LIN {X 0,Y 220.797,Z 443.981,A -85,B 0,C 180,E1 -20381.946,E2 -20381.946} C_VEL
LIN {X 0,Y 220.875,Z 443.967,A -85,B 0,C 180,E1 -20387.041,E2 -20387.041} C_VEL
LIN {X 0,Y 220.861,Z 443.966,A -85,B 0,C 180,E1 -20390.474,E2 -20390.474} C_VEL
LIN {X 0,Y 220.818,Z 443.975,A -85,B 0,C 180,E1 -20395.048,E2 -20395.048} C_VEL
LIN {X 0,Y 220.906,Z 444.135,A -85,B 0,C 180,E1 -20396.999,E2 -20396.999} C_VEL
LIN {X 0,Y 221.881,Z 446.769,A -85,B 0,C 180,E1 -20397.42,E2 -20397.42} C_VEL
LIN {X 0,Y 226.651,Z 456.679,A -85,B 0,C 180,E1 -20399.386,E2 -20399.386} C_VEL
LIN {X 0,Y 230.145,Z 465.491,A -85,B 0,C 180,E1 -20401.214,E2 -20401.214} C_VEL
LIN {X 0,Y 233.063,Z 475.055,A -85,B 0,C 180,E1 -20403.323,E2 -20403.323} C_VEL
LIN {X 0,Y 234.867,Z 483.039,A -85,B 0,C 180,E1 -20405.233,E2 -20405.233} C_VEL
LIN {X 0,Y 232.591,Z 492.857,A -85,B 0,C 180,E1 -20407.34,E2 -20407.34} C_VEL
LIN {X 0,Y 230.039,Z 502.346,A -85,B 0,C 180,E1 -20409.897,E2 -20409.897} C_VEL
LIN {X 0,Y 227.751,Z 509.911,A -85,B 0,C 180,E1 -20412.49,E2 -20412.49} C_VEL
LIN {X 0,Y 226.25,Z 515.061,A -85,B 0,C 180,E1 -20414.7,E2 -20414.7} C_VEL
LIN {X 0,Y 224.746,Z 520.013,A -85,B 0,C 180,E1 -20417.356,E2 -20417.356} C_VEL
LIN {X 0,Y 223.377,Z 523.89,A -85,B 0,C 180,E1 -20420.035,E2 -20420.035} C_VEL
LIN {X 0,Y 222.303,Z 526.757,A -85,B 0,C 180,E1 -20422.735,E2 -20422.735} C_VEL
LIN {X 0,Y 221.792,Z 528.126,A -85,B 0,C 180,E1 -20424.545,E2 -20424.545} C_VEL
LIN {X 0,Y 221.55,Z 529.649,A -85,B 0,C 180,E1 -20428.182,E2 -20428.182} C_VEL
LIN {X 0,Y 221.511,Z 529.869,A -85,B 0,C 180,E1 -20430,E2 -20430} C_VEL
LIN {X 0,Y 221.549,Z 529.683,A -85,B 0,C 180,E1 -20431.818,E2 -20431.818} C_VEL
LIN {X 0,Y 221.782,Z 528.204,A -85,B 0,C 180,E1 -20435.455,E2 -20435.455} C_VEL
LIN {X 0,Y 222.287,Z 526.871,A -85,B 0,C 180,E1 -20437.265,E2 -20437.265} C_VEL
LIN {X 0,Y 223.365,Z 524.046,A -85,B 0,C 180,E1 -20439.965,E2 -20439.965} C_VEL
LIN {X 0,Y 224.708,Z 520.225,A -85,B 0,C 180,E1 -20442.646,E2 -20442.646} C_VEL
LIN {X 0,Y 226.414,Z 514.308,A -85,B 0,C 180,E1 -20445.791,E2 -20445.791} C_VEL
LIN {X 0,Y 228.461,Z 507.907,A -85,B 0,C 180,E1 -20448.38,E2 -20448.38} C_VEL
LIN {X 0,Y 230.832,Z 499.865,A -85,B 0,C 180,E1 -20450.962,E2 -20450.962} C_VEL
LIN {X 0,Y 232.897,Z 491.636,A -85,B 0,C 180,E1 -20453.097,E2 -20453.097} C_VEL
LIN {X 0,Y 234.818,Z 483.666,A -85,B 0,C 180,E1 -20454.772,E2 -20454.772} C_VEL
LIN {X 0,Y 234.22,Z 479.238,A -85,B 0,C 180,E1 -20455.818,E2 -20455.818} C_VEL
LIN {X 0,Y 231.252,Z 468.913,A -85,B 0,C 180,E1 -20458.195,E2 -20458.195} C_VEL
LIN {X 0,Y 227.759,Z 459.239,A -85,B 0,C 180,E1 -20460.231,E2 -20460.231} C_VEL
LIN {X 0,Y 222.646,Z 448.097,A -85,B 0,C 180,E1 -20462.454,E2 -20462.454} C_VEL
LIN {X 0,Y 220.923,Z 444.348,A -85,B 0,C 180,E1 -20463.132,E2 -20463.132} C_VEL
LIN {X 0,Y 220.874,Z 443.97,A -85,B 0,C 180,E1 -20463.221,E2 -20463.221} C_VEL
LIN {X 0,Y 220.869,Z 443.973,A -85,B 0,C 180,E1 -20467.298,E2 -20467.298} C_VEL
LIN {X 0,Y 220.873,Z 443.971,A -85,B 0,C 180,E1 -20471.929,E2 -20471.929} C_VEL
LIN {X 0,Y 220.792,Z 443.981,A -85,B 0,C 180,E1 -20475.55,E2 -20475.55} C_VEL
LIN {X 0,Y 220.811,Z 443.98,A -85,B 0,C 180,E1 -20480.464,E2 -20480.464} C_VEL
LIN {X 0,Y 220.802,Z 443.984,A -85,B 0,C 180,E1 -20485.045,E2 -20485.045} C_VEL
LIN {X 0,Y 220.835,Z 443.977,A -85,B 0,C 180,E1 -20489.39,E2 -20489.39} C_VEL
LIN {X 0,Y 220.896,Z 443.967,A -85,B 0,C 180,E1 -20493.549,E2 -20493.549} C_VEL
LIN {X 0,Y 220.88,Z 443.963,A -85,B 0,C 180,E1 -20497.553,E2 -20497.553} C_VEL
LIN {X 0,Y 220.986,Z 443.952,A -85,B 0,C 180,E1 -20502.571,E2 -20502.571} C_VEL
LIN {X 0,Y 221.014,Z 443.95,A -85,B 0,C 180,E1 -20507.139,E2 -20507.139} C_VEL
LIN {X 0,Y 221.204,Z 443.931,A -85,B 0,C 180,E1 -20510.859,E2 -20510.859} C_VEL
LIN {X 0,Y 221.14,Z 443.925,A -85,B 0,C 180,E1 -20514.529,E2 -20514.529} C_VEL
LIN {X 0,Y 221.515,Z 443.892,A -85,B 0,C 180,E1 -20518.182,E2 -20518.182} C_VEL
LIN {X 0,Y 221.515,Z 443.88,A -85,B 0,C 180,E1 -20521.818,E2 -20521.818} C_VEL
LIN {X 0,Y 221.257,Z 443.916,A -85,B 0,C 180,E1 -20527.299,E2 -20527.299} C_VEL
LIN {X 0,Y 221.083,Z 443.944,A -85,B 0,C 180,E1 -20530.996,E2 -20530.996} C_VEL
LIN {X 0,Y 221.018,Z 443.949,A -85,B 0,C 180,E1 -20536.63,E2 -20536.63} C_VEL
LIN {X 0,Y 220.886,Z 443.973,A -85,B 0,C 180,E1 -20540.487,E2 -20540.487} C_VEL
LIN {X 0,Y 220.863,Z 443.975,A -85,B 0,C 180,E1 -20544.435,E2 -20544.435} C_VEL
LIN {X 0,Y 220.828,Z 443.978,A -85,B 0,C 180,E1 -20548.515,E2 -20548.515} C_VEL
LIN {X 0,Y 220.83,Z 444.003,A -85,B 0,C 180,E1 -20551.675,E2 -20551.675} C_VEL
LIN {X 0,Y 221.956,Z 449.045,A -85,B 0,C 180,E1 -20555.858,E2 -20555.858} C_VEL
LIN {X 0,Y 223.004,Z 454.546,A -85,B 0,C 180,E1 -20560.02,E2 -20560.02} C_VEL
LIN {X 0,Y 224.02,Z 459.907,A -85,B 0,C 180,E1 -20563.816,E2 -20563.816} C_VEL
LIN {X 0,Y 225.122,Z 465.25,A -85,B 0,C 180,E1 -20567.382,E2 -20567.382} C_VEL
LIN {X 0,Y 225.601,Z 467.977,A -85,B 0,C 180,E1 -20569.141,E2 -20569.141} C_VEL
LIN {X 0,Y 225.692,Z 469.86,A -85,B 0,C 180,E1 -20570.314,E2 -20570.314} C_VEL
LIN {X 0,Y 224.095,Z 476.513,A -85,B 0,C 180,E1 -20574.172,E2 -20574.172} C_VEL
LIN {X 0,Y 223.25,Z 479.952,A -85,B 0,C 180,E1 -20576.149,E2 -20576.149} C_VEL
LIN {X 0,Y 224.695,Z 487.159,A -85,B 0,C 180,E1 -20576.76,E2 -20576.76} C_VEL
LIN {X 0,Y 226.787,Z 499.616,A -85,B 0,C 180,E1 -20577.987,E2 -20577.987} C_VEL
LIN {X 0,Y 228.055,Z 512.378,A -85,B 0,C 180,E1 -20579.46,E2 -20579.46} C_VEL
LIN {X 0,Y 228.416,Z 525.424,A -85,B 0,C 180,E1 -20581.265,E2 -20581.265} C_VEL
LIN {X 0,Y 228.421,Z 526.853,A -85,B 0,C 180,E1 -20581.483,E2 -20581.483} C_VEL
LIN {X 0,Y 227.726,Z 531.904,A -85,B 0,C 180,E1 -20582.228,E2 -20582.228} C_VEL
LIN {X 0,Y 225.999,Z 536.833,A -85,B 0,C 180,E1 -20582.945,E2 -20582.945} C_VEL
LIN {X 0,Y 220.98,Z 547.697,A -85,B 0,C 180,E1 -20584.798,E2 -20584.798} C_VEL
LIN {X 0,Y 219.703,Z 552.067,A -85,B 0,C 180,E1 -20585.794,E2 -20585.794} C_VEL
LIN {X 0,Y 218.356,Z 559.465,A -85,B 0,C 180,E1 -20587.779,E2 -20587.779} C_VEL
LIN {X 0,Y 215.907,Z 568.5,A -85,B 0,C 180,E1 -20590.732,E2 -20590.732} C_VEL
LIN {X 0,Y 214.238,Z 574.791,A -85,B 0,C 180,E1 -20593.319,E2 -20593.319} C_VEL
LIN {X 0,Y 213.015,Z 581.157,A -85,B 0,C 180,E1 -20596.647,E2 -20596.647} C_VEL
LIN {X 0,Y 212.567,Z 585.353,A -85,B 0,C 180,E1 -20599.523,E2 -20599.523} C_VEL
LIN {X 0,Y 212.669,Z 588.586,A -85,B 0,C 180,E1 -20602.481,E2 -20602.481} C_VEL
LIN {X 0,Y 213.218,Z 591.167,A -85,B 0,C 180,E1 -20606.22,E2 -20606.22} C_VEL
LIN {X 0,Y 213.999,Z 592.157,A -85,B 0,C 180,E1 -20610,E2 -20610} C_VEL
LIN {X 0,Y 213.215,Z 591.15,A -85,B 0,C 180,E1 -20613.78,E2 -20613.78} C_VEL
LIN {X 0,Y 212.627,Z 588.624,A -85,B 0,C 180,E1 -20617.432,E2 -20617.432} C_VEL
LIN {X 0,Y 212.568,Z 585.304,A -85,B 0,C 180,E1 -20620.477,E2 -20620.477} C_VEL
LIN {X 0,Y 213.014,Z 581.088,A -85,B 0,C 180,E1 -20623.353,E2 -20623.353} C_VEL
LIN {X 0,Y 214.21,Z 574.691,A -85,B 0,C 180,E1 -20626.683,E2 -20626.683} C_VEL
LIN {X 0,Y 215.907,Z 568.382,A -85,B 0,C 180,E1 -20629.269,E2 -20629.269} C_VEL
LIN {X 0,Y 218.348,Z 559.319,A -85,B 0,C 180,E1 -20632.222,E2 -20632.222} C_VEL
LIN {X 0,Y 219.865,Z 550.517,A -85,B 0,C 180,E1 -20634.554,E2 -20634.554} C_VEL
LIN {X 0,Y 221.04,Z 540.018,A -85,B 0,C 180,E1 -20636.856,E2 -20636.856} C_VEL
LIN {X 0,Y 221.682,Z 528.784,A -85,B 0,C 180,E1 -20638.913,E2 -20638.913} C_VEL
LIN {X 0,Y 221.703,Z 517.176,A -85,B 0,C 180,E1 -20640.699,E2 -20640.699} C_VEL
LIN {X 0,Y 220.89,Z 504.818,A -85,B 0,C 180,E1 -20642.312,E2 -20642.312} C_VEL
LIN {X 0,Y 219.065,Z 491.67,A -85,B 0,C 180,E1 -20643.777,E2 -20643.777} C_VEL
LIN {X 0,Y 216.635,Z 478.749,A -85,B 0,C 180,E1 -20645.03,E2 -20645.03} C_VEL
LIN {X 0,Y 218.558,Z 471.281,A -85,B 0,C 180,E1 -20649.489,E2 -20649.489} C_VEL
LIN {X 0,Y 218.545,Z 468.802,A -85,B 0,C 180,E1 -20651.076,E2 -20651.076} C_VEL
LIN {X 0,Y 217.309,Z 462.5,A -85,B 0,C 180,E1 -20655.358,E2 -20655.358} C_VEL
LIN {X 0,Y 216.224,Z 456.823,A -85,B 0,C 180,E1 -20659.453,E2 -20659.453} C_VEL
LIN {X 0,Y 215.145,Z 450.979,A -85,B 0,C 180,E1 -20663.985,E2 -20663.985} C_VEL
LIN {X 0,Y 213.875,Z 445.272,A -85,B 0,C 180,E1 -20668.917,E2 -20668.917} C_VEL
LIN {X 0,Y 213.779,Z 444.857,A -85,B 0,C 180,E1 -20669.56,E2 -20669.56} C_VEL
LIN {X 0,Y 213.828,Z 444.855,A -85,B 0,C 180,E1 -20672.604,E2 -20672.604} C_VEL
LIN {X 0,Y 213.822,Z 444.849,A -85,B 0,C 180,E1 -20676.974,E2 -20676.974} C_VEL
LIN {X 0,Y 213.947,Z 444.836,A -85,B 0,C 180,E1 -20682.804,E2 -20682.804} C_VEL
LIN {X 0,Y 213.957,Z 444.837,A -85,B 0,C 180,E1 -20686.707,E2 -20686.707} C_VEL
LIN {X 0,Y 214.142,Z 444.811,A -85,B 0,C 180,E1 -20690.555,E2 -20690.555} C_VEL
LIN {X 0,Y 214.103,Z 444.817,A -85,B 0,C 180,E1 -20694.349,E2 -20694.349} C_VEL
LIN {X 0,Y 214.45,Z 444.774,A -85,B 0,C 180,E1 -20698.122,E2 -20698.122} C_VEL
LIN {X 0,Y 214.558,Z 444.757,A -85,B 0,C 180,E1 -20700,E2 -20700} C_VEL
LIN {X 0,Y 214.449,Z 444.773,A -85,B 0,C 180,E1 -20701.878,E2 -20701.878} C_VEL
LIN {X 0,Y 214.197,Z 444.802,A -85,B 0,C 180,E1 -20707.542,E2 -20707.542} C_VEL
LIN {X 0,Y 214.011,Z 444.816,A -85,B 0,C 180,E1 -20711.364,E2 -20711.364} C_VEL
LIN {X 0,Y 213.936,Z 444.787,A -85,B 0,C 180,E1 -20715.237,E2 -20715.237} C_VEL
LIN {X 0,Y 213.843,Z 444.831,A -85,B 0,C 180,E1 -20719.187,E2 -20719.187} C_VEL
LIN {X 0,Y 213.85,Z 444.841,A -85,B 0,C 180,E1 -20723.227,E2 -20723.227} C_VEL
LIN {X 0,Y 213.832,Z 444.809,A -85,B 0,C 180,E1 -20727.45,E2 -20727.45} C_VEL
LIN {X 0,Y 213.77,Z 444.852,A -85,B 0,C 180,E1 -20731.737,E2 -20731.737} C_VEL
LIN {X 0,Y 213.746,Z 444.855,A -85,B 0,C 180,E1 -20736.288,E2 -20736.288} C_VEL
LIN {X 0,Y 213.728,Z 444.861,A -85,B 0,C 180,E1 -20741.122,E2 -20741.122} C_VEL
LIN {X 0,Y 213.75,Z 444.854,A -85,B 0,C 180,E1 -20743.668,E2 -20743.668} C_VEL
LIN {X 0,Y 213.814,Z 444.85,A -85,B 0,C 180,E1 -20746.349,E2 -20746.349} C_VEL
LIN {X 0,Y 213.8,Z 444.851,A -85,B 0,C 180,E1 -20749.118,E2 -20749.118} C_VEL
LIN {X 0,Y 213.759,Z 444.849,A -85,B 0,C 180,E1 -20753.714,E2 -20753.714} C_VEL
LIN {X 0,Y 213.799,Z 445.01,A -85,B 0,C 180,E1 -20755.719,E2 -20755.719} C_VEL
LIN {X 0,Y 214.42,Z 446.987,A -85,B 0,C 180,E1 -20756.032,E2 -20756.032} C_VEL
LIN {X 0,Y 215.693,Z 448.943,A -85,B 0,C 180,E1 -20756.485,E2 -20756.485} C_VEL
LIN {X 0,Y 220.507,Z 459.407,A -85,B 0,C 180,E1 -20758.674,E2 -20758.674} C_VEL
LIN {X 0,Y 224.284,Z 469.275,A -85,B 0,C 180,E1 -20760.865,E2 -20760.865} C_VEL
LIN {X 0,Y 227.226,Z 479.67,A -85,B 0,C 180,E1 -20763.327,E2 -20763.327} C_VEL
LIN {X 0,Y 228.28,Z 485.103,A -85,B 0,C 180,E1 -20764.712,E2 -20764.712} C_VEL
LIN {X 0,Y 226.124,Z 493.865,A -85,B 0,C 180,E1 -20766.654,E2 -20766.654} C_VEL
LIN {X 0,Y 223.452,Z 503.353,A -85,B 0,C 180,E1 -20769.278,E2 -20769.278} C_VEL
LIN {X 0,Y 221.059,Z 510.918,A -85,B 0,C 180,E1 -20771.942,E2 -20771.942} C_VEL
LIN {X 0,Y 219.481,Z 516.063,A -85,B 0,C 180,E1 -20774.213,E2 -20774.213} C_VEL
LIN {X 0,Y 217.895,Z 521.019,A -85,B 0,C 180,E1 -20776.951,E2 -20776.951} C_VEL
LIN {X 0,Y 216.458,Z 524.896,A -85,B 0,C 180,E1 -20779.713,E2 -20779.713} C_VEL
LIN {X 0,Y 215.333,Z 527.763,A -85,B 0,C 180,E1 -20782.498,E2 -20782.498} C_VEL
LIN {X 0,Y 214.797,Z 529.132,A -85,B 0,C 180,E1 -20784.367,E2 -20784.367} C_VEL
LIN {X 0,Y 214.526,Z 530.654,A -85,B 0,C 180,E1 -20788.122,E2 -20788.122} C_VEL
LIN {X 0,Y 214.484,Z 530.874,A -85,B 0,C 180,E1 -20790,E2 -20790} C_VEL
LIN {X 0,Y 214.525,Z 530.687,A -85,B 0,C 180,E1 -20791.877,E2 -20791.877} C_VEL
LIN {X 0,Y 214.787,Z 529.209,A -85,B 0,C 180,E1 -20795.633,E2 -20795.633} C_VEL
LIN {X 0,Y 215.317,Z 527.875,A -85,B 0,C 180,E1 -20797.502,E2 -20797.502} C_VEL
LIN {X 0,Y 216.446,Z 525.05,A -85,B 0,C 180,E1 -20800.287,E2 -20800.287} C_VEL
LIN {X 0,Y 217.856,Z 521.229,A -85,B 0,C 180,E1 -20803.051,E2 -20803.051} C_VEL
LIN {X 0,Y 219.658,Z 515.315,A -85,B 0,C 180,E1 -20806.288,E2 -20806.288} C_VEL
LIN {X 0,Y 221.803,Z 508.91,A -85,B 0,C 180,E1 -20808.952,E2 -20808.952} C_VEL
LIN {X 0,Y 224.283,Z 500.868,A -85,B 0,C 180,E1 -20811.604,E2 -20811.604} C_VEL
LIN {X 0,Y 226.451,Z 492.638,A -85,B 0,C 180,E1 -20813.795,E2 -20813.795} C_VEL
LIN {X 0,Y 228.303,Z 484.691,A -85,B 0,C 180,E1 -20815.529,E2 -20815.529} C_VEL
LIN {X 0,Y 226.822,Z 477.955,A -85,B 0,C 180,E1 -20817.232,E2 -20817.232} C_VEL
LIN {X 0,Y 224.28,Z 469.314,A -85,B 0,C 180,E1 -20819.278,E2 -20819.278} C_VEL
LIN {X 0,Y 220.91,Z 460.371,A -85,B 0,C 180,E1 -20821.272,E2 -20821.272} C_VEL
LIN {X 0,Y 215.802,Z 449.254,A -85,B 0,C 180,E1 -20823.617,E2 -20823.617} C_VEL
LIN {X 0,Y 213.944,Z 445.703,A -85,B 0,C 180,E1 -20824.345,E2 -20824.345} C_VEL
LIN {X 0,Y 213.773,Z 444.851,A -85,B 0,C 180,E1 -20824.476,E2 -20824.476} C_VEL
LIN {X 0,Y 213.805,Z 444.853,A -85,B 0,C 180,E1 -20828.649,E2 -20828.649} C_VEL
LIN {X 0,Y 213.829,Z 444.851,A -85,B 0,C 180,E1 -20831.098,E2 -20831.098} C_VEL
LIN {X 0,Y 213.81,Z 444.851,A -85,B 0,C 180,E1 -20833.685,E2 -20833.685} C_VEL
LIN {X 0,Y 213.749,Z 444.86,A -85,B 0,C 180,E1 -20836.332,E2 -20836.332} C_VEL
LIN {X 0,Y 213.727,Z 444.863,A -85,B 0,C 180,E1 -20841.334,E2 -20841.334} C_VEL
LIN {X 0,Y 213.758,Z 444.859,A -85,B 0,C 180,E1 -20846.018,E2 -20846.018} C_VEL
LIN {X 0,Y 213.762,Z 444.86,A -85,B 0,C 180,E1 -20850.451,E2 -20850.451} C_VEL
LIN {X 0,Y 213.803,Z 444.854,A -85,B 0,C 180,E1 -20854.702,E2 -20854.702} C_VEL
LIN {X 0,Y 213.815,Z 444.848,A -85,B 0,C 180,E1 -20858.803,E2 -20858.803} C_VEL
LIN {X 0,Y 213.946,Z 444.828,A -85,B 0,C 180,E1 -20862.804,E2 -20862.804} C_VEL
LIN {X 0,Y 213.956,Z 444.831,A -85,B 0,C 180,E1 -20866.707,E2 -20866.707} C_VEL
LIN {X 0,Y 214.142,Z 444.811,A -85,B 0,C 180,E1 -20870.555,E2 -20870.555} C_VEL
LIN {X 0,Y 214.1,Z 444.802,A -85,B 0,C 180,E1 -20874.348,E2 -20874.348} C_VEL
LIN {X 0,Y 214.448,Z 444.772,A -85,B 0,C 180,E1 -20878.122,E2 -20878.122} C_VEL
LIN {X 0,Y 214.557,Z 444.756,A -85,B 0,C 180,E1 -20880,E2 -20880} C_VEL
LIN {X 0,Y 214.448,Z 444.76,A -85,B 0,C 180,E1 -20881.878,E2 -20881.878} C_VEL
LIN {X 0,Y 214.196,Z 444.794,A -85,B 0,C 180,E1 -20887.541,E2 -20887.541} C_VEL
LIN {X 0,Y 214.01,Z 444.825,A -85,B 0,C 180,E1 -20891.364,E2 -20891.364} C_VEL
LIN {X 0,Y 213.936,Z 444.836,A -85,B 0,C 180,E1 -20895.237,E2 -20895.237} C_VEL
LIN {X 0,Y 213.838,Z 444.849,A -85,B 0,C 180,E1 -20899.187,E2 -20899.187} C_VEL
LIN {X 0,Y 213.812,Z 444.852,A -85,B 0,C 180,E1 -20903.231,E2 -20903.231} C_VEL
LIN {X 0,Y 213.83,Z 444.85,A -85,B 0,C 180,E1 -20907.45,E2 -20907.45} C_VEL
LIN {X 0,Y 213.81,Z 445.01,A -85,B 0,C 180,E1 -20910.769,E2 -20910.769} C_VEL
LIN {X 0,Y 214.585,Z 448.483,A -85,B 0,C 180,E1 -20913.833,E2 -20913.833} C_VEL
LIN {X 0,Y 215.7,Z 453.941,A -85,B 0,C 180,E1 -20918.248,E2 -20918.248} C_VEL
LIN {X 0,Y 216.85,Z 460.139,A -85,B 0,C 180,E1 -20922.891,E2 -20922.891} C_VEL
LIN {X 0,Y 218.259,Z 467.186,A -85,B 0,C 180,E1 -20927.783,E2 -20927.783} C_VEL
LIN {X 0,Y 218.664,Z 470.579,A -85,B 0,C 180,E1 -20929.998,E2 -20929.998} C_VEL
LIN {X 0,Y 217.389,Z 475.884,A -85,B 0,C 180,E1 -20933.204,E2 -20933.204} C_VEL
LIN {X 0,Y 216.645,Z 478.821,A -85,B 0,C 180,E1 -20934.965,E2 -20934.965} C_VEL
LIN {X 0,Y 219.458,Z 493.611,A -85,B 0,C 180,E1 -20936.37,E2 -20936.37} C_VEL
LIN {X 0,Y 221.046,Z 505.767,A -85,B 0,C 180,E1 -20937.754,E2 -20937.754} C_VEL
LIN {X 0,Y 221.758,Z 517.676,A -85,B 0,C 180,E1 -20939.327,E2 -20939.327} C_VEL
LIN {X 0,Y 221.762,Z 529.086,A -85,B 0,C 180,E1 -20941.099,E2 -20941.099} C_VEL
LIN {X 0,Y 221.056,Z 540.207,A -85,B 0,C 180,E1 -20943.136,E2 -20943.136} C_VEL
LIN {X 0,Y 219.923,Z 550.713,A -85,B 0,C 180,E1 -20945.453,E2 -20945.453} C_VEL
LIN {X 0,Y 219.703,Z 552.067,A -85,B 0,C 180,E1 -20945.794,E2 -20945.794} C_VEL
LIN {X 0,Y 218.282,Z 556.263,A -85,B 0,C 180,E1 -20946.832,E2 -20946.832} C_VEL
LIN {X 0,Y 215.837,Z 560.132,A -85,B 0,C 180,E1 -20947.837,E2 -20947.837} C_VEL
LIN {X 0,Y 209.492,Z 568.242,A -85,B 0,C 180,E1 -20950.383,E2 -20950.383} C_VEL
LIN {X 0,Y 207.939,Z 571.438,A -85,B 0,C 180,E1 -20951.691,E2 -20951.691} C_VEL
LIN {X 0,Y 206.73,Z 576.698,A -85,B 0,C 180,E1 -20954.219,E2 -20954.219} C_VEL
LIN {X 0,Y 205.804,Z 581.639,A -85,B 0,C 180,E1 -20957.175,E2 -20957.175} C_VEL
LIN {X 0,Y 205.483,Z 585.478,A -85,B 0,C 180,E1 -20960.153,E2 -20960.153} C_VEL
LIN {X 0,Y 205.589,Z 587.76,A -85,B 0,C 180,E1 -20962.463,E2 -20962.463} C_VEL
LIN {X 0,Y 206.151,Z 590.155,A -85,B 0,C 180,E1 -20966.091,E2 -20966.091} C_VEL
LIN {X 0,Y 206.959,Z 591.15,A -85,B 0,C 180,E1 -20970,E2 -20970} C_VEL
LIN {X 0,Y 206.146,Z 590.137,A -85,B 0,C 180,E1 -20973.91,E2 -20973.91} C_VEL
LIN {X 0,Y 205.579,Z 587.744,A -85,B 0,C 180,E1 -20977.518,E2 -20977.518} C_VEL
LIN {X 0,Y 205.54,Z 584.28,A -85,B 0,C 180,E1 -20980.84,E2 -20980.84} C_VEL
LIN {X 0,Y 206.04,Z 580.06,A -85,B 0,C 180,E1 -20983.814,E2 -20983.814} C_VEL
LIN {X 0,Y 207.35,Z 573.664,A -85,B 0,C 180,E1 -20987.252,E2 -20987.252} C_VEL
LIN {X 0,Y 209.32,Z 566.787,A -85,B 0,C 180,E1 -20990.13,E2 -20990.13} C_VEL
LIN {X 0,Y 211.678,Z 558.283,A -85,B 0,C 180,E1 -20992.962,E2 -20992.962} C_VEL
LIN {X 0,Y 213.201,Z 549.463,A -85,B 0,C 180,E1 -20995.375,E2 -20995.375} C_VEL
LIN {X 0,Y 214.448,Z 538.887,A -85,B 0,C 180,E1 -20997.766,E2 -20997.766} C_VEL
LIN {X 0,Y 215.125,Z 527.761,A -85,B 0,C 180,E1 -20999.871,E2 -20999.871} C_VEL
LIN {X 0,Y 215.164,Z 515.163,A -85,B 0,C 180,E1 -21001.87,E2 -21001.87} C_VEL
LIN {X 0,Y 214.282,Z 503.326,A -85,B 0,C 180,E1 -21003.474,E2 -21003.474} C_VEL
LIN {X 0,Y 212.397,Z 489.867,A -85,B 0,C 180,E1 -21005.038,E2 -21005.038} C_VEL
LIN {X 0,Y 210.128,Z 478.735,A -85,B 0,C 180,E1 -21006.159,E2 -21006.159} C_VEL
LIN {X 0,Y 210.063,Z 477.645,A -85,B 0,C 180,E1 -21006.277,E2 -21006.277} C_VEL
LIN {X 0,Y 211.333,Z 472.954,A -85,B 0,C 180,E1 -21009.188,E2 -21009.188} C_VEL
LIN {X 0,Y 211.566,Z 470.402,A -85,B 0,C 180,E1 -21010.833,E2 -21010.833} C_VEL
LIN {X 0,Y 210.624,Z 465.201,A -85,B 0,C 180,E1 -21014.485,E2 -21014.485} C_VEL
LIN {X 0,Y 209.391,Z 458.887,A -85,B 0,C 180,E1 -21019.118,E2 -21019.118} C_VEL
LIN {X 0,Y 208.279,Z 452.737,A -85,B 0,C 180,E1 -21024.081,E2 -21024.081} C_VEL
LIN {X 0,Y 207.308,Z 448.347,A -85,B 0,C 180,E1 -21027.945,E2 -21027.945} C_VEL
LIN {X 0,Y 206.736,Z 445.739,A -85,B 0,C 180,E1 -21030.467,E2 -21030.467} C_VEL
LIN {X 0,Y 206.733,Z 445.734,A -85,B 0,C 180,E1 -21033.772,E2 -21033.772} C_VEL
LIN {X 0,Y 206.741,Z 445.726,A -85,B 0,C 180,E1 -21038.041,E2 -21038.041} C_VEL
LIN {X 0,Y 206.876,Z 445.718,A -85,B 0,C 180,E1 -21042.197,E2 -21042.197} C_VEL
LIN {X 0,Y 206.899,Z 445.717,A -85,B 0,C 180,E1 -21046.245,E2 -21046.245} C_VEL
LIN {X 0,Y 207.102,Z 445.689,A -85,B 0,C 180,E1 -21050.231,E2 -21050.231} C_VEL
LIN {X 0,Y 207.064,Z 445.694,A -85,B 0,C 180,E1 -21054.156,E2 -21054.156} C_VEL
LIN {X 0,Y 207.386,Z 445.654,A -85,B 0,C 180,E1 -21058.058,E2 -21058.058} C_VEL
LIN {X 0,Y 207.522,Z 445.634,A -85,B 0,C 180,E1 -21060,E2 -21060} C_VEL
LIN {X 0,Y 207.385,Z 445.653,A -85,B 0,C 180,E1 -21061.942,E2 -21061.942} C_VEL
LIN {X 0,Y 207.14,Z 445.682,A -85,B 0,C 180,E1 -21067.8,E2 -21067.8} C_VEL
LIN {X 0,Y 206.935,Z 445.694,A -85,B 0,C 180,E1 -21071.758,E2 -21071.758} C_VEL
LIN {X 0,Y 206.869,Z 445.664,A -85,B 0,C 180,E1 -21075.771,E2 -21075.771} C_VEL
LIN {X 0,Y 206.787,Z 445.715,A -85,B 0,C 180,E1 -21079.869,E2 -21079.869} C_VEL
LIN {X 0,Y 206.766,Z 445.719,A -85,B 0,C 180,E1 -21084.072,E2 -21084.072} C_VEL
LIN {X 0,Y 206.739,Z 445.692,A -85,B 0,C 180,E1 -21088.42,E2 -21088.42} C_VEL
LIN {X 0,Y 206.701,Z 445.736,A -85,B 0,C 180,E1 -21092.958,E2 -21092.958} C_VEL
LIN {X 0,Y 206.683,Z 445.739,A -85,B 0,C 180,E1 -21097.74,E2 -21097.74} C_VEL
LIN {X 0,Y 206.66,Z 445.743,A -85,B 0,C 180,E1 -21101.568,E2 -21101.568} C_VEL
LIN {X 0,Y 206.711,Z 445.736,A -85,B 0,C 180,E1 -21105.56,E2 -21105.56} C_VEL
LIN {X 0,Y 206.73,Z 445.728,A -85,B 0,C 180,E1 -21109.764,E2 -21109.764} C_VEL
LIN {X 0,Y 206.709,Z 445.729,A -85,B 0,C 180,E1 -21114.305,E2 -21114.305} C_VEL
LIN {X 0,Y 207.069,Z 447.238,A -85,B 0,C 180,E1 -21114.545,E2 -21114.545} C_VEL
LIN {X 0,Y 211.704,Z 456.085,A -85,B 0,C 180,E1 -21116.545,E2 -21116.545} C_VEL
LIN {X 0,Y 216.246,Z 466.752,A -85,B 0,C 180,E1 -21119.001,E2 -21119.001} C_VEL
LIN {X 0,Y 219.329,Z 476.127,A -85,B 0,C 180,E1 -21121.272,E2 -21121.272} C_VEL
LIN {X 0,Y 221.539,Z 485.16,A -85,B 0,C 180,E1 -21123.632,E2 -21123.632} C_VEL
LIN {X 0,Y 221.693,Z 487.159,A -85,B 0,C 180,E1 -21124.157,E2 -21124.157} C_VEL
LIN {X 0,Y 219.206,Z 496.618,A -85,B 0,C 180,E1 -21126.374,E2 -21126.374} C_VEL
LIN {X 0,Y 216.894,Z 504.361,A -85,B 0,C 180,E1 -21128.621,E2 -21128.621} C_VEL
LIN {X 0,Y 214.388,Z 511.925,A -85,B 0,C 180,E1 -21131.36,E2 -21131.36} C_VEL
LIN {X 0,Y 212.729,Z 517.065,A -85,B 0,C 180,E1 -21133.696,E2 -21133.696} C_VEL
LIN {X 0,Y 211.055,Z 522.025,A -85,B 0,C 180,E1 -21136.52,E2 -21136.52} C_VEL
LIN {X 0,Y 209.548,Z 525.902,A -85,B 0,C 180,E1 -21139.37,E2 -21139.37} C_VEL
LIN {X 0,Y 208.367,Z 528.769,A -85,B 0,C 180,E1 -21142.246,E2 -21142.246} C_VEL
LIN {X 0,Y 207.804,Z 530.137,A -85,B 0,C 180,E1 -21144.177,E2 -21144.177} C_VEL
LIN {X 0,Y 207.503,Z 531.659,A -85,B 0,C 180,E1 -21148.059,E2 -21148.059} C_VEL
LIN {X 0,Y 207.458,Z 531.879,A -85,B 0,C 180,E1 -21150,E2 -21150} C_VEL
LIN {X 0,Y 207.502,Z 531.692,A -85,B 0,C 180,E1 -21151.941,E2 -21151.941} C_VEL
LIN {X 0,Y 207.794,Z 530.214,A -85,B 0,C 180,E1 -21155.823,E2 -21155.823} C_VEL
LIN {X 0,Y 208.351,Z 528.88,A -85,B 0,C 180,E1 -21157.754,E2 -21157.754} C_VEL
LIN {X 0,Y 209.535,Z 526.055,A -85,B 0,C 180,E1 -21160.63,E2 -21160.63} C_VEL
LIN {X 0,Y 211.015,Z 522.233,A -85,B 0,C 180,E1 -21163.482,E2 -21163.482} C_VEL
LIN {X 0,Y 212.929,Z 516.301,A -85,B 0,C 180,E1 -21166.826,E2 -21166.826} C_VEL
LIN {X 0,Y 215.558,Z 508.713,A -85,B 0,C 180,E1 -21170.019,E2 -21170.019} C_VEL
LIN {X 0,Y 218.204,Z 500.339,A -85,B 0,C 180,E1 -21172.737,E2 -21172.737} C_VEL
LIN {X 0,Y 220.531,Z 491.744,A -85,B 0,C 180,E1 -21174.977,E2 -21174.977} C_VEL
LIN {X 0,Y 221.831,Z 486.725,A -85,B 0,C 180,E1 -21176.077,E2 -21176.077} C_VEL
LIN {X 0,Y 219.909,Z 478.148,A -85,B 0,C 180,E1 -21178.358,E2 -21178.358} C_VEL
LIN {X 0,Y 216.833,Z 468.197,A -85,B 0,C 180,E1 -21180.806,E2 -21180.806} C_VEL
LIN {X 0,Y 212.935,Z 458.816,A -85,B 0,C 180,E1 -21183.01,E2 -21183.01} C_VEL
LIN {X 0,Y 208.357,Z 449.431,A -85,B 0,C 180,E1 -21185.118,E2 -21185.118} C_VEL
LIN {X 0,Y 206.897,Z 446.699,A -85,B 0,C 180,E1 -21185.712,E2 -21185.712} C_VEL
LIN {X 0,Y 206.709,Z 445.736,A -85,B 0,C 180,E1 -21185.907,E2 -21185.907} C_VEL
LIN {X 0,Y 206.753,Z 445.731,A -85,B 0,C 180,E1 -21190.23,E2 -21190.23} C_VEL
LIN {X 0,Y 206.71,Z 445.733,A -85,B 0,C 180,E1 -21194.439,E2 -21194.439} C_VEL
LIN {X 0,Y 206.669,Z 445.741,A -85,B 0,C 180,E1 -21199.75,E2 -21199.75} C_VEL
LIN {X 0,Y 206.7,Z 445.738,A -85,B 0,C 180,E1 -21204.689,E2 -21204.689} C_VEL
LIN {X 0,Y 206.708,Z 445.738,A -85,B 0,C 180,E1 -21209.336,E2 -21209.336} C_VEL
LIN {X 0,Y 206.734,Z 445.731,A -85,B 0,C 180,E1 -21213.772,E2 -21213.772} C_VEL
LIN {X 0,Y 206.759,Z 445.722,A -85,B 0,C 180,E1 -21218.043,E2 -21218.043} C_VEL
LIN {X 0,Y 206.878,Z 445.71,A -85,B 0,C 180,E1 -21222.197,E2 -21222.197} C_VEL
LIN {X 0,Y 206.898,Z 445.714,A -85,B 0,C 180,E1 -21226.244,E2 -21226.244} C_VEL
LIN {X 0,Y 207.101,Z 445.686,A -85,B 0,C 180,E1 -21230.231,E2 -21230.231} C_VEL
LIN {X 0,Y 207.061,Z 445.679,A -85,B 0,C 180,E1 -21234.156,E2 -21234.156} C_VEL
LIN {X 0,Y 207.384,Z 445.651,A -85,B 0,C 180,E1 -21238.058,E2 -21238.058} C_VEL
LIN {X 0,Y 207.521,Z 445.631,A -85,B 0,C 180,E1 -21240,E2 -21240} C_VEL
LIN {X 0,Y 207.385,Z 445.639,A -85,B 0,C 180,E1 -21241.942,E2 -21241.942} C_VEL
LIN {X 0,Y 207.139,Z 445.673,A -85,B 0,C 180,E1 -21247.8,E2 -21247.8} C_VEL
LIN {X 0,Y 206.933,Z 445.704,A -85,B 0,C 180,E1 -21251.758,E2 -21251.758} C_VEL
LIN {X 0,Y 206.87,Z 445.716,A -85,B 0,C 180,E1 -21255.77,E2 -21255.77} C_VEL
LIN {X 0,Y 206.78,Z 445.728,A -85,B 0,C 180,E1 -21259.869,E2 -21259.869} C_VEL
LIN {X 0,Y 206.748,Z 445.734,A -85,B 0,C 180,E1 -21264.074,E2 -21264.074} C_VEL
LIN {X 0,Y 206.738,Z 445.734,A -85,B 0,C 180,E1 -21268.42,E2 -21268.42} C_VEL
LIN {X 0,Y 206.744,Z 445.866,A -85,B 0,C 180,E1 -21269.672,E2 -21269.672} C_VEL
LIN {X 0,Y 207.779,Z 450.508,A -85,B 0,C 180,E1 -21273.925,E2 -21273.925} C_VEL
LIN {X 0,Y 208.843,Z 455.782,A -85,B 0,C 180,E1 -21278.338,E2 -21278.338} C_VEL
LIN {X 0,Y 210.072,Z 462.407,A -85,B 0,C 180,E1 -21283.414,E2 -21283.414} C_VEL
LIN {X 0,Y 211.111,Z 467.504,A -85,B 0,C 180,E1 -21287.087,E2 -21287.087} C_VEL
LIN {X 0,Y 211.637,Z 471.469,A -85,B 0,C 180,E1 -21289.799,E2 -21289.799} C_VEL
LIN {X 0,Y 210.353,Z 476.628,A -85,B 0,C 180,E1 -21293.031,E2 -21293.031} C_VEL
LIN {X 0,Y 210.079,Z 477.781,A -85,B 0,C 180,E1 -21293.718,E2 -21293.718} C_VEL
LIN {X 0,Y 211.395,Z 484.35,A -85,B 0,C 180,E1 -21294.33,E2 -21294.33} C_VEL
LIN {X 0,Y 213.689,Z 497.561,A -85,B 0,C 180,E1 -21295.778,E2 -21295.778} C_VEL
LIN {X 0,Y 214.907,Z 509.391,A -85,B 0,C 180,E1 -21297.271,E2 -21297.271} C_VEL
LIN {X 0,Y 215.31,Z 521.672,A -85,B 0,C 180,E1 -21299.071,E2 -21299.071} C_VEL
LIN {X 0,Y 214.948,Z 533.515,A -85,B 0,C 180,E1 -21301.131,E2 -21301.131} C_VEL
LIN {X 0,Y 213.865,Z 544.522,A -85,B 0,C 180,E1 -21303.401,E2 -21303.401} C_VEL
LIN {X 0,Y 212.672,Z 553.378,A -85,B 0,C 180,E1 -21305.602,E2 -21305.602} C_VEL
LIN {X 0,Y 210.87,Z 561.484,A -85,B 0,C 180,E1 -21307.979,E2 -21307.979} C_VEL
LIN {X 0,Y 208.502,Z 569.555,A -85,B 0,C 180,E1 -21310.9,E2 -21310.9} C_VEL
LIN {X 0,Y 207.939,Z 571.438,A -85,B 0,C 180,E1 -21311.691,E2 -21311.691} C_VEL
LIN {X 0,Y 206.534,Z 574.447,A -85,B 0,C 180,E1 -21313.058,E2 -21313.058} C_VEL
LIN {X 0,Y 201.177,Z 580.102,A -85,B 0,C 180,E1 -21316.291,E2 -21316.291} C_VEL
LIN {X 0,Y 198.861,Z 582.767,A -85,B 0,C 180,E1 -21318.318,E2 -21318.318} C_VEL
LIN {X 0,Y 198.454,Z 583.997,A -85,B 0,C 180,E1 -21319.39,E2 -21319.39} C_VEL
LIN {X 0,Y 198.53,Z 586.9,A -85,B 0,C 180,E1 -21322.397,E2 -21322.397} C_VEL
LIN {X 0,Y 199.063,Z 589.139,A -85,B 0,C 180,E1 -21325.951,E2 -21325.951} C_VEL
LIN {X 0,Y 199.918,Z 590.143,A -85,B 0,C 180,E1 -21330,E2 -21330} C_VEL
LIN {X 0,Y 199.056,Z 589.12,A -85,B 0,C 180,E1 -21334.049,E2 -21334.049} C_VEL
LIN {X 0,Y 198.505,Z 586.906,A -85,B 0,C 180,E1 -21337.55,E2 -21337.55} C_VEL
LIN {X 0,Y 198.501,Z 583.253,A -85,B 0,C 180,E1 -21341.229,E2 -21341.229} C_VEL
LIN {X 0,Y 199.078,Z 579.033,A -85,B 0,C 180,E1 -21344.307,E2 -21344.307} C_VEL
LIN {X 0,Y 200.506,Z 572.635,A -85,B 0,C 180,E1 -21347.861,E2 -21347.861} C_VEL
LIN {X 0,Y 202.6,Z 565.759,A -85,B 0,C 180,E1 -21350.828,E2 -21350.828} C_VEL
LIN {X 0,Y 204.664,Z 558.783,A -85,B 0,C 180,E1 -21353.26,E2 -21353.26} C_VEL
LIN {X 0,Y 206.286,Z 550.288,A -85,B 0,C 180,E1 -21355.746,E2 -21355.746} C_VEL
LIN {X 0,Y 207.591,Z 540.678,A -85,B 0,C 180,E1 -21358.1,E2 -21358.1} C_VEL
LIN {X 0,Y 208.423,Z 530.991,A -85,B 0,C 180,E1 -21360.105,E2 -21360.105} C_VEL
LIN {X 0,Y 208.765,Z 520.154,A -85,B 0,C 180,E1 -21362.026,E2 -21362.026} C_VEL
LIN {X 0,Y 208.416,Z 508.838,A -85,B 0,C 180,E1 -21363.75,E2 -21363.75} C_VEL
LIN {X 0,Y 206.935,Z 495.199,A -85,B 0,C 180,E1 -21365.55,E2 -21365.55} C_VEL
LIN {X 0,Y 204.717,Z 482.683,A -85,B 0,C 180,E1 -21366.985,E2 -21366.985} C_VEL
LIN {X 0,Y 203.522,Z 476.519,A -85,B 0,C 180,E1 -21367.64,E2 -21367.64} C_VEL
LIN {X 0,Y 204.368,Z 473.62,A -85,B 0,C 180,E1 -21369.509,E2 -21369.509} C_VEL
LIN {X 0,Y 204.582,Z 471.52,A -85,B 0,C 180,E1 -21370.907,E2 -21370.907} C_VEL
LIN {X 0,Y 203.552,Z 465.976,A -85,B 0,C 180,E1 -21374.944,E2 -21374.944} C_VEL
LIN {X 0,Y 202.318,Z 459.617,A -85,B 0,C 180,E1 -21379.838,E2 -21379.838} C_VEL
LIN {X 0,Y 201.499,Z 455.05,A -85,B 0,C 180,E1 -21383.634,E2 -21383.634} C_VEL
LIN {X 0,Y 200.412,Z 449.949,A -85,B 0,C 180,E1 -21388.263,E2 -21388.263} C_VEL
LIN {X 0,Y 199.71,Z 446.609,A -85,B 0,C 180,E1 -21391.616,E2 -21391.616} C_VEL
LIN {X 0,Y 199.717,Z 446.603,A -85,B 0,C 180,E1 -21397.227,E2 -21397.227} C_VEL
LIN {X 0,Y 199.799,Z 446.599,A -85,B 0,C 180,E1 -21401.758,E2 -21401.758} C_VEL
LIN {X 0,Y 199.839,Z 446.595,A -85,B 0,C 180,E1 -21405.749,E2 -21405.749} C_VEL
LIN {X 0,Y 200.025,Z 446.573,A -85,B 0,C 180,E1 -21409.882,E2 -21409.882} C_VEL
LIN {X 0,Y 200.025,Z 446.57,A -85,B 0,C 180,E1 -21413.949,E2 -21413.949} C_VEL
LIN {X 0,Y 200.325,Z 446.534,A -85,B 0,C 180,E1 -21417.99,E2 -21417.99} C_VEL
LIN {X 0,Y 200.486,Z 446.51,A -85,B 0,C 180,E1 -21420,E2 -21420} C_VEL
LIN {X 0,Y 200.03,Z 446.567,A -85,B 0,C 180,E1 -21424.03,E2 -21424.03} C_VEL
LIN {X 0,Y 200.089,Z 446.561,A -85,B 0,C 180,E1 -21428.077,E2 -21428.077} C_VEL
LIN {X 0,Y 199.882,Z 446.568,A -85,B 0,C 180,E1 -21432.179,E2 -21432.179} C_VEL
LIN {X 0,Y 199.807,Z 446.543,A -85,B 0,C 180,E1 -21436.343,E2 -21436.343} C_VEL
LIN {X 0,Y 199.703,Z 446.602,A -85,B 0,C 180,E1 -21440.605,E2 -21440.605} C_VEL
LIN {X 0,Y 199.675,Z 446.591,A -85,B 0,C 180,E1 -21444.984,E2 -21444.984} C_VEL
LIN {X 0,Y 199.667,Z 446.581,A -85,B 0,C 180,E1 -21449.524,E2 -21449.524} C_VEL
LIN {X 0,Y 199.674,Z 446.609,A -85,B 0,C 180,E1 -21452.355,E2 -21452.355} C_VEL
LIN {X 0,Y 199.625,Z 446.615,A -85,B 0,C 180,E1 -21456.763,E2 -21456.763} C_VEL
LIN {X 0,Y 199.614,Z 446.614,A -85,B 0,C 180,E1 -21459.327,E2 -21459.327} C_VEL
LIN {X 0,Y 199.6,Z 446.622,A -85,B 0,C 180,E1 -21462.318,E2 -21462.318} C_VEL
LIN {X 0,Y 199.648,Z 446.616,A -85,B 0,C 180,E1 -21465.248,E2 -21465.248} C_VEL
LIN {X 0,Y 199.67,Z 446.608,A -85,B 0,C 180,E1 -21468.028,E2 -21468.028} C_VEL
LIN {X 0,Y 199.682,Z 446.604,A -85,B 0,C 180,E1 -21472.796,E2 -21472.796} C_VEL
LIN {X 0,Y 200.687,Z 449.458,A -85,B 0,C 180,E1 -21473.351,E2 -21473.351} C_VEL
LIN {X 0,Y 205.523,Z 458.527,A -85,B 0,C 180,E1 -21475.585,E2 -21475.585} C_VEL
LIN {X 0,Y 209.872,Z 468.93,A -85,B 0,C 180,E1 -21478.136,E2 -21478.136} C_VEL
LIN {X 0,Y 212.636,Z 477.229,A -85,B 0,C 180,E1 -21480.279,E2 -21480.279} C_VEL
LIN {X 0,Y 214.834,Z 486.238,A -85,B 0,C 180,E1 -21482.742,E2 -21482.742} C_VEL
LIN {X 0,Y 215.243,Z 488.835,A -85,B 0,C 180,E1 -21483.49,E2 -21483.49} C_VEL
LIN {X 0,Y 212.788,Z 497.626,A -85,B 0,C 180,E1 -21485.616,E2 -21485.616} C_VEL
LIN {X 0,Y 210.365,Z 505.368,A -85,B 0,C 180,E1 -21487.923,E2 -21487.923} C_VEL
LIN {X 0,Y 207.741,Z 512.932,A -85,B 0,C 180,E1 -21490.74,E2 -21490.74} C_VEL
LIN {X 0,Y 205.994,Z 518.069,A -85,B 0,C 180,E1 -21493.146,E2 -21493.146} C_VEL
LIN {X 0,Y 204.227,Z 523.032,A -85,B 0,C 180,E1 -21496.061,E2 -21496.061} C_VEL
LIN {X 0,Y 202.645,Z 526.908,A -85,B 0,C 180,E1 -21499.003,E2 -21499.003} C_VEL
LIN {X 0,Y 201.406,Z 529.774,A -85,B 0,C 180,E1 -21501.976,E2 -21501.976} C_VEL
LIN {X 0,Y 200.813,Z 531.143,A -85,B 0,C 180,E1 -21503.973,E2 -21503.973} C_VEL
LIN {X 0,Y 200.48,Z 532.664,A -85,B 0,C 180,E1 -21507.991,E2 -21507.991} C_VEL
LIN {X 0,Y 200.431,Z 532.884,A -85,B 0,C 180,E1 -21510,E2 -21510} C_VEL
LIN {X 0,Y 200.479,Z 532.697,A -85,B 0,C 180,E1 -21512.009,E2 -21512.009} C_VEL
LIN {X 0,Y 200.803,Z 531.218,A -85,B 0,C 180,E1 -21516.027,E2 -21516.027} C_VEL
LIN {X 0,Y 201.389,Z 529.885,A -85,B 0,C 180,E1 -21518.024,E2 -21518.024} C_VEL
LIN {X 0,Y 202.632,Z 527.059,A -85,B 0,C 180,E1 -21520.997,E2 -21520.997} C_VEL
LIN {X 0,Y 204.188,Z 523.237,A -85,B 0,C 180,E1 -21523.942,E2 -21523.942} C_VEL
LIN {X 0,Y 206.21,Z 517.309,A -85,B 0,C 180,E1 -21527.39,E2 -21527.39} C_VEL
LIN {X 0,Y 208.559,Z 510.916,A -85,B 0,C 180,E1 -21530.206,E2 -21530.206} C_VEL
LIN {X 0,Y 211.279,Z 502.873,A -85,B 0,C 180,E1 -21533.008,E2 -21533.008} C_VEL
LIN {X 0,Y 213.671,Z 494.641,A -85,B 0,C 180,E1 -21535.315,E2 -21535.315} C_VEL
LIN {X 0,Y 215.275,Z 488.798,A -85,B 0,C 180,E1 -21536.666,E2 -21536.666} C_VEL
LIN {X 0,Y 213.944,Z 482.085,A -85,B 0,C 180,E1 -21538.569,E2 -21538.569} C_VEL
LIN {X 0,Y 211.499,Z 473.361,A -85,B 0,C 180,E1 -21540.878,E2 -21540.878} C_VEL
LIN {X 0,Y 207.732,Z 463.554,A -85,B 0,C 180,E1 -21543.359,E2 -21543.359} C_VEL
LIN {X 0,Y 203.308,Z 454.016,A -85,B 0,C 180,E1 -21545.674,E2 -21545.674} C_VEL
LIN {X 0,Y 199.994,Z 447.917,A -85,B 0,C 180,E1 -21547.146,E2 -21547.146} C_VEL
LIN {X 0,Y 199.709,Z 446.608,A -85,B 0,C 180,E1 -21547.409,E2 -21547.409} C_VEL
LIN {X 0,Y 199.687,Z 446.611,A -85,B 0,C 180,E1 -21551.967,E2 -21551.967} C_VEL
LIN {X 0,Y 199.632,Z 446.614,A -85,B 0,C 180,E1 -21555.243,E2 -21555.243} C_VEL
LIN {X 0,Y 199.599,Z 446.62,A -85,B 0,C 180,E1 -21558.01,E2 -21558.01} C_VEL
LIN {X 0,Y 199.616,Z 446.622,A -85,B 0,C 180,E1 -21560.766,E2 -21560.766} C_VEL
LIN {X 0,Y 199.614,Z 446.621,A -85,B 0,C 180,E1 -21565.713,E2 -21565.713} C_VEL
LIN {X 0,Y 199.694,Z 446.604,A -85,B 0,C 180,E1 -21568.136,E2 -21568.136} C_VEL
LIN {X 0,Y 199.687,Z 446.605,A -85,B 0,C 180,E1 -21572.772,E2 -21572.772} C_VEL
LIN {X 0,Y 199.74,Z 446.596,A -85,B 0,C 180,E1 -21577.229,E2 -21577.229} C_VEL
LIN {X 0,Y 199.839,Z 446.589,A -85,B 0,C 180,E1 -21581.722,E2 -21581.722} C_VEL
LIN {X 0,Y 199.838,Z 446.592,A -85,B 0,C 180,E1 -21585.748,E2 -21585.748} C_VEL
LIN {X 0,Y 200.024,Z 446.566,A -85,B 0,C 180,E1 -21589.882,E2 -21589.882} C_VEL
LIN {X 0,Y 200.023,Z 446.556,A -85,B 0,C 180,E1 -21593.949,E2 -21593.949} C_VEL
LIN {X 0,Y 200.324,Z 446.53,A -85,B 0,C 180,E1 -21597.989,E2 -21597.989} C_VEL
LIN {X 0,Y 200.485,Z 446.507,A -85,B 0,C 180,E1 -21600,E2 -21600} C_VEL
LIN {X 0,Y 200.031,Z 446.566,A -85,B 0,C 180,E1 -21604.029,E2 -21604.029} C_VEL
LIN {X 0,Y 200.088,Z 446.551,A -85,B 0,C 180,E1 -21608.077,E2 -21608.077} C_VEL
LIN {X 0,Y 199.881,Z 446.58,A -85,B 0,C 180,E1 -21612.179,E2 -21612.179} C_VEL
LIN {X 0,Y 199.807,Z 446.591,A -85,B 0,C 180,E1 -21616.343,E2 -21616.343} C_VEL
LIN {X 0,Y 199.692,Z 446.613,A -85,B 0,C 180,E1 -21620.606,E2 -21620.606} C_VEL
LIN {X 0,Y 199.666,Z 446.615,A -85,B 0,C 180,E1 -21624.985,E2 -21624.985} C_VEL
LIN {X 0,Y 199.717,Z 446.737,A -85,B 0,C 180,E1 -21628.515,E2 -21628.515} C_VEL
LIN {X 0,Y 200.724,Z 451.217,A -85,B 0,C 180,E1 -21632.826,E2 -21632.826} C_VEL
LIN {X 0,Y 201.783,Z 456.585,A -85,B 0,C 180,E1 -21637.569,E2 -21637.569} C_VEL
LIN {X 0,Y 202.851,Z 462.506,A -85,B 0,C 180,E1 -21642.316,E2 -21642.316} C_VEL
LIN {X 0,Y 203.943,Z 467.933,A -85,B 0,C 180,E1 -21646.432,E2 -21646.432} C_VEL
LIN {X 0,Y 204.595,Z 471.879,A -85,B 0,C 180,E1 -21649.257,E2 -21649.257} C_VEL
LIN {X 0,Y 203.896,Z 475.504,A -85,B 0,C 180,E1 -21651.652,E2 -21651.652} C_VEL
LIN {X 0,Y 203.572,Z 476.562,A -85,B 0,C 180,E1 -21652.329,E2 -21652.329} C_VEL
LIN {X 0,Y 204.357,Z 480.431,A -85,B 0,C 180,E1 -21652.723,E2 -21652.723} C_VEL
LIN {X 0,Y 206.925,Z 494.467,A -85,B 0,C 180,E1 -21654.311,E2 -21654.311} C_VEL
LIN {X 0,Y 208.353,Z 507.47,A -85,B 0,C 180,E1 -21656.004,E2 -21656.004} C_VEL
LIN {X 0,Y 208.822,Z 520.304,A -85,B 0,C 180,E1 -21657.949,E2 -21657.949} C_VEL
LIN {X 0,Y 208.396,Z 532.629,A -85,B 0,C 180,E1 -21660.17,E2 -21660.17} C_VEL
LIN {X 0,Y 207.323,Z 543.474,A -85,B 0,C 180,E1 -21662.492,E2 -21662.492} C_VEL
LIN {X 0,Y 206.023,Z 552.333,A -85,B 0,C 180,E1 -21664.76,E2 -21664.76} C_VEL
LIN {X 0,Y 204.269,Z 560.465,A -85,B 0,C 180,E1 -21667.228,E2 -21667.228} C_VEL
LIN {X 0,Y 202.071,Z 567.727,A -85,B 0,C 180,E1 -21669.894,E2 -21669.894} C_VEL
LIN {X 0,Y 200.263,Z 573.774,A -85,B 0,C 180,E1 -21672.645,E2 -21672.645} C_VEL
LIN {X 0,Y 199.082,Z 579.107,A -85,B 0,C 180,E1 -21675.693,E2 -21675.693} C_VEL
LIN {X 0,Y 198.454,Z 583.997,A -85,B 0,C 180,E1 -21679.39,E2 -21679.39} C_VEL
LIN {X 0,Y 197.758,Z 585.634,A -85,B 0,C 180,E1 -21681.021,E2 -21681.021} C_VEL
LIN {X 0,Y 195.092,Z 587.485,A -85,B 0,C 180,E1 -21683.756,E2 -21683.756} C_VEL
LIN {X 0,Y 193.023,Z 588.385,A -85,B 0,C 180,E1 -21686.024,E2 -21686.024} C_VEL
LIN {X 0,Y 192.352,Z 588.802,A -85,B 0,C 180,E1 -21687.783,E2 -21687.783} C_VEL
LIN {X 0,Y 192.409,Z 588.895,A -85,B 0,C 180,E1 -21688.375,E2 -21688.375} C_VEL
LIN {X 0,Y 192.875,Z 589.136,A -85,B 0,C 180,E1 -21690,E2 -21690} C_VEL
LIN {X 0,Y 191.952,Z 588.101,A -85,B 0,C 180,E1 -21694.2,E2 -21694.2} C_VEL
LIN {X 0,Y 191.445,Z 586.047,A -85,B 0,C 180,E1 -21697.616,E2 -21697.616} C_VEL
LIN {X 0,Y 191.489,Z 582.229,A -85,B 0,C 180,E1 -21701.646,E2 -21701.646} C_VEL
LIN {X 0,Y 192.133,Z 578.005,A -85,B 0,C 180,E1 -21704.836,E2 -21704.836} C_VEL
LIN {X 0,Y 193.688,Z 571.608,A -85,B 0,C 180,E1 -21708.512,E2 -21708.512} C_VEL
LIN {X 0,Y 195.928,Z 564.733,A -85,B 0,C 180,E1 -21711.572,E2 -21711.572} C_VEL
LIN {X 0,Y 198.036,Z 557.745,A -85,B 0,C 180,E1 -21714.087,E2 -21714.087} C_VEL
LIN {X 0,Y 199.676,Z 549.232,A -85,B 0,C 180,E1 -21716.665,E2 -21716.665} C_VEL
LIN {X 0,Y 201.101,Z 539.55,A -85,B 0,C 180,E1 -21719.109,E2 -21719.109} C_VEL
LIN {X 0,Y 202.019,Z 528.515,A -85,B 0,C 180,E1 -21721.456,E2 -21721.456} C_VEL
LIN {X 0,Y 202.313,Z 516.977,A -85,B 0,C 180,E1 -21723.517,E2 -21723.517} C_VEL
LIN {X 0,Y 201.732,Z 504.863,A -85,B 0,C 180,E1 -21725.395,E2 -21725.395} C_VEL
LIN {X 0,Y 200.182,Z 491.725,A -85,B 0,C 180,E1 -21727.171,E2 -21727.171} C_VEL
LIN {X 0,Y 197.783,Z 479.011,A -85,B 0,C 180,E1 -21728.68,E2 -21728.68} C_VEL
LIN {X 0,Y 197.068,Z 475.421,A -85,B 0,C 180,E1 -21729.075,E2 -21729.075} C_VEL
LIN {X 0,Y 197.565,Z 473.049,A -85,B 0,C 180,E1 -21730.697,E2 -21730.697} C_VEL
LIN {X 0,Y 196.734,Z 468.064,A -85,B 0,C 180,E1 -21734.4,E2 -21734.4} C_VEL
LIN {X 0,Y 195.459,Z 461.47,A -85,B 0,C 180,E1 -21739.668,E2 -21739.668} C_VEL
LIN {X 0,Y 194.651,Z 456.865,A -85,B 0,C 180,E1 -21743.591,E2 -21743.591} C_VEL
LIN {X 0,Y 193.59,Z 451.897,A -85,B 0,C 180,E1 -21748.237,E2 -21748.237} C_VEL
LIN {X 0,Y 192.637,Z 447.496,A -85,B 0,C 180,E1 -21752.868,E2 -21752.868} C_VEL
LIN {X 0,Y 192.687,Z 447.485,A -85,B 0,C 180,E1 -21756.346,E2 -21756.346} C_VEL
LIN {X 0,Y 192.734,Z 447.478,A -85,B 0,C 180,E1 -21761.458,E2 -21761.458} C_VEL
LIN {X 0,Y 192.767,Z 447.476,A -85,B 0,C 180,E1 -21765.214,E2 -21765.214} C_VEL
LIN {X 0,Y 192.947,Z 447.456,A -85,B 0,C 180,E1 -21769.567,E2 -21769.567} C_VEL
LIN {X 0,Y 192.987,Z 447.447,A -85,B 0,C 180,E1 -21773.728,E2 -21773.728} C_VEL
LIN {X 0,Y 193.267,Z 447.413,A -85,B 0,C 180,E1 -21777.916,E2 -21777.916} C_VEL
LIN {X 0,Y 193.45,Z 447.386,A -85,B 0,C 180,E1 -21780,E2 -21780} C_VEL
LIN {X 0,Y 192.976,Z 447.447,A -85,B 0,C 180,E1 -21784.177,E2 -21784.177} C_VEL
LIN {X 0,Y 193.037,Z 447.439,A -85,B 0,C 180,E1 -21788.374,E2 -21788.374} C_VEL
LIN {X 0,Y 192.808,Z 447.44,A -85,B 0,C 180,E1 -21792.633,E2 -21792.633} C_VEL
LIN {X 0,Y 192.76,Z 447.423,A -85,B 0,C 180,E1 -21796.959,E2 -21796.959} C_VEL
LIN {X 0,Y 192.64,Z 447.485,A -85,B 0,C 180,E1 -21801.397,E2 -21801.397} C_VEL
LIN {X 0,Y 192.667,Z 447.472,A -85,B 0,C 180,E1 -21804.225,E2 -21804.225} C_VEL
LIN {X 0,Y 192.647,Z 447.446,A -85,B 0,C 180,E1 -21808.889,E2 -21808.889} C_VEL
LIN {X 0,Y 192.599,Z 447.494,A -85,B 0,C 180,E1 -21813.186,E2 -21813.186} C_VEL
LIN {X 0,Y 192.555,Z 447.499,A -85,B 0,C 180,E1 -21818.351,E2 -21818.351} C_VEL
LIN {X 0,Y 192.541,Z 447.497,A -85,B 0,C 180,E1 -21823.111,E2 -21823.111} C_VEL
LIN {X 0,Y 192.603,Z 447.487,A -85,B 0,C 180,E1 -21826.869,E2 -21826.869} C_VEL
LIN {X 0,Y 192.673,Z 447.569,A -85,B 0,C 180,E1 -21831.177,E2 -21831.177} C_VEL
LIN {X 0,Y 193.678,Z 450.32,A -85,B 0,C 180,E1 -21831.746,E2 -21831.746} C_VEL
LIN {X 0,Y 194.639,Z 451.577,A -85,B 0,C 180,E1 -21832.132,E2 -21832.132} C_VEL
LIN {X 0,Y 199.855,Z 462.035,A -85,B 0,C 180,E1 -21834.847,E2 -21834.847} C_VEL
LIN {X 0,Y 203.912,Z 472.172,A -85,B 0,C 180,E1 -21837.522,E2 -21837.522} C_VEL
LIN {X 0,Y 206.67,Z 480.91,A -85,B 0,C 180,E1 -21839.94,E2 -21839.94} C_VEL
LIN {X 0,Y 208.508,Z 489.056,A -85,B 0,C 180,E1 -21842.329,E2 -21842.329} C_VEL
LIN {X 0,Y 208.747,Z 490.402,A -85,B 0,C 180,E1 -21842.738,E2 -21842.738} C_VEL
LIN {X 0,Y 206.41,Z 498.633,A -85,B 0,C 180,E1 -21844.81,E2 -21844.81} C_VEL
LIN {X 0,Y 203.87,Z 506.376,A -85,B 0,C 180,E1 -21847.181,E2 -21847.181} C_VEL
LIN {X 0,Y 201.12,Z 513.939,A -85,B 0,C 180,E1 -21850.08,E2 -21850.08} C_VEL
LIN {X 0,Y 199.28,Z 519.074,A -85,B 0,C 180,E1 -21852.559,E2 -21852.559} C_VEL
LIN {X 0,Y 197.414,Z 524.038,A -85,B 0,C 180,E1 -21855.569,E2 -21855.569} C_VEL
LIN {X 0,Y 195.751,Z 527.914,A -85,B 0,C 180,E1 -21858.611,E2 -21858.611} C_VEL
LIN {X 0,Y 194.449,Z 530.78,A -85,B 0,C 180,E1 -21861.687,E2 -21861.687} C_VEL
LIN {X 0,Y 193.826,Z 532.149,A -85,B 0,C 180,E1 -21863.755,E2 -21863.755} C_VEL
LIN {X 0,Y 193.457,Z 533.669,A -85,B 0,C 180,E1 -21867.918,E2 -21867.918} C_VEL
LIN {X 0,Y 193.404,Z 533.889,A -85,B 0,C 180,E1 -21870,E2 -21870} C_VEL
LIN {X 0,Y 193.456,Z 533.702,A -85,B 0,C 180,E1 -21872.082,E2 -21872.082} C_VEL
LIN {X 0,Y 193.815,Z 532.223,A -85,B 0,C 180,E1 -21876.245,E2 -21876.245} C_VEL
LIN {X 0,Y 194.432,Z 530.889,A -85,B 0,C 180,E1 -21878.313,E2 -21878.313} C_VEL
LIN {X 0,Y 195.738,Z 528.063,A -85,B 0,C 180,E1 -21881.389,E2 -21881.389} C_VEL
LIN {X 0,Y 197.374,Z 524.241,A -85,B 0,C 180,E1 -21884.433,E2 -21884.433} C_VEL
LIN {X 0,Y 199.513,Z 518.316,A -85,B 0,C 180,E1 -21887.991,E2 -21887.991} C_VEL
LIN {X 0,Y 201.978,Z 511.919,A -85,B 0,C 180,E1 -21890.895,E2 -21890.895} C_VEL
LIN {X 0,Y 204.829,Z 503.876,A -85,B 0,C 180,E1 -21893.776,E2 -21893.776} C_VEL
LIN {X 0,Y 207.345,Z 495.642,A -85,B 0,C 180,E1 -21896.144,E2 -21896.144} C_VEL
LIN {X 0,Y 208.75,Z 490.761,A -85,B 0,C 180,E1 -21897.321,E2 -21897.321} C_VEL
LIN {X 0,Y 207.556,Z 484.249,A -85,B 0,C 180,E1 -21899.254,E2 -21899.254} C_VEL
LIN {X 0,Y 204.766,Z 474.353,A -85,B 0,C 180,E1 -21902.038,E2 -21902.038} C_VEL
LIN {X 0,Y 200.88,Z 464.48,A -85,B 0,C 180,E1 -21904.695,E2 -21904.695} C_VEL
LIN {X 0,Y 196.304,Z 454.951,A -85,B 0,C 180,E1 -21907.194,E2 -21907.194} C_VEL
LIN {X 0,Y 192.953,Z 448.778,A -85,B 0,C 180,E1 -21908.793,E2 -21908.793} C_VEL
LIN {X 0,Y 192.685,Z 447.484,A -85,B 0,C 180,E1 -21909.086,E2 -21909.086} C_VEL
LIN {X 0,Y 192.599,Z 447.493,A -85,B 0,C 180,E1 -21913.893,E2 -21913.893} C_VEL
LIN {X 0,Y 192.527,Z 447.498,A -85,B 0,C 180,E1 -21918.923,E2 -21918.923} C_VEL
LIN {X 0,Y 192.588,Z 447.491,A -85,B 0,C 180,E1 -21923.402,E2 -21923.402} C_VEL
LIN {X 0,Y 192.609,Z 447.487,A -85,B 0,C 180,E1 -21927.059,E2 -21927.059} C_VEL
LIN {X 0,Y 192.662,Z 447.481,A -85,B 0,C 180,E1 -21931.691,E2 -21931.691} C_VEL
LIN {X 0,Y 192.708,Z 447.477,A -85,B 0,C 180,E1 -21936.349,E2 -21936.349} C_VEL
LIN {X 0,Y 192.783,Z 447.468,A -85,B 0,C 180,E1 -21941.414,E2 -21941.414} C_VEL
LIN {X 0,Y 192.767,Z 447.473,A -85,B 0,C 180,E1 -21945.214,E2 -21945.214} C_VEL
LIN {X 0,Y 192.946,Z 447.447,A -85,B 0,C 180,E1 -21949.567,E2 -21949.567} C_VEL
LIN {X 0,Y 192.985,Z 447.433,A -85,B 0,C 180,E1 -21953.728,E2 -21953.728} C_VEL
LIN {X 0,Y 193.265,Z 447.409,A -85,B 0,C 180,E1 -21957.916,E2 -21957.916} C_VEL
LIN {X 0,Y 193.449,Z 447.383,A -85,B 0,C 180,E1 -21960,E2 -21960} C_VEL
LIN {X 0,Y 192.977,Z 447.445,A -85,B 0,C 180,E1 -21964.177,E2 -21964.177} C_VEL
LIN {X 0,Y 193.036,Z 447.43,A -85,B 0,C 180,E1 -21968.374,E2 -21968.374} C_VEL
LIN {X 0,Y 192.807,Z 447.459,A -85,B 0,C 180,E1 -21972.633,E2 -21972.633} C_VEL
LIN {X 0,Y 192.76,Z 447.467,A -85,B 0,C 180,E1 -21976.958,E2 -21976.958} C_VEL
LIN {X 0,Y 192.624,Z 447.492,A -85,B 0,C 180,E1 -21981.399,E2 -21981.399} C_VEL
LIN {X 0,Y 192.649,Z 447.49,A -85,B 0,C 180,E1 -21984.213,E2 -21984.213} C_VEL
LIN {X 0,Y 192.659,Z 447.622,A -85,B 0,C 180,E1 -21987.275,E2 -21987.275} C_VEL
LIN {X 0,Y 193.917,Z 453.204,A -85,B 0,C 180,E1 -21992.931,E2 -21992.931} C_VEL
LIN {X 0,Y 194.955,Z 458.578,A -85,B 0,C 180,E1 -21997.795,E2 -21997.795} C_VEL
LIN {X 0,Y 196.081,Z 464.775,A -85,B 0,C 180,E1 -22002.922,E2 -22002.922} C_VEL
LIN {X 0,Y 197.203,Z 470.527,A -85,B 0,C 180,E1 -22007.38,E2 -22007.38} C_VEL
LIN {X 0,Y 197.536,Z 473.134,A -85,B 0,C 180,E1 -22009.302,E2 -22009.302} C_VEL
LIN {X 0,Y 197.116,Z 475.668,A -85,B 0,C 180,E1 -22010.91,E2 -22010.91} C_VEL
LIN {X 0,Y 200.064,Z 490.213,A -85,B 0,C 180,E1 -22012.588,E2 -22012.588} C_VEL
LIN {X 0,Y 201.753,Z 503.835,A -85,B 0,C 180,E1 -22014.405,E2 -22014.405} C_VEL
LIN {X 0,Y 202.343,Z 515.839,A -85,B 0,C 180,E1 -22016.239,E2 -22016.239} C_VEL
LIN {X 0,Y 202.161,Z 527.702,A -85,B 0,C 180,E1 -22018.345,E2 -22018.345} C_VEL
LIN {X 0,Y 201.354,Z 537.896,A -85,B 0,C 180,E1 -22020.461,E2 -22020.461} C_VEL
LIN {X 0,Y 199.991,Z 547.555,A -85,B 0,C 180,E1 -22022.817,E2 -22022.817} C_VEL
LIN {X 0,Y 198.413,Z 556.364,A -85,B 0,C 180,E1 -22025.405,E2 -22025.405} C_VEL
LIN {X 0,Y 196.357,Z 563.598,A -85,B 0,C 180,E1 -22027.925,E2 -22027.925} C_VEL
LIN {X 0,Y 194.019,Z 570.67,A -85,B 0,C 180,E1 -22030.973,E2 -22030.973} C_VEL
LIN {X 0,Y 192.544,Z 576.421,A -85,B 0,C 180,E1 -22034.112,E2 -22034.112} C_VEL
LIN {X 0,Y 191.625,Z 580.979,A -85,B 0,C 180,E1 -22037.288,E2 -22037.288} C_VEL
LIN {X 0,Y 191.358,Z 584.479,A -85,B 0,C 180,E1 -22040.487,E2 -22040.487} C_VEL
LIN {X 0,Y 191.584,Z 586.988,A -85,B 0,C 180,E1 -22043.682,E2 -22043.682} C_VEL
LIN {X 0,Y 191.96,Z 588.121,A -85,B 0,C 180,E1 -22045.801,E2 -22045.801} C_VEL
LIN {X 0,Y 192.409,Z 588.895,A -85,B 0,C 180,E1 -22048.375,E2 -22048.375} C_VEL
LIN {X 0,Y 192.264,Z 589.02,A -85,B 0,C 180,E1 -22049.538,E2 -22049.538} C_VEL
LIN {X 0,Y 191.46,Z 588.884,A -85,B 0,C 180,E1 -22050.685,E2 -22050.685} C_VEL
LIN {X 0,Y 188.762,Z 588.112,A -85,B 0,C 180,E1 -22052.931,E2 -22052.931} C_VEL
LIN {X 0,Y 185.837,Z 586.851,A -85,B 0,C 180,E1 -22055.235,E2 -22055.235} C_VEL
LIN {X 0,Y 184.51,Z 585.666,A -85,B 0,C 180,E1 -22057.036,E2 -22057.036} C_VEL
LIN {X 0,Y 184.375,Z 585.211,A -85,B 0,C 180,E1 -22057.652,E2 -22057.652} C_VEL
LIN {X 0,Y 184.362,Z 582.356,A -85,B 0,C 180,E1 -22060.988,E2 -22060.988} C_VEL
LIN {X 0,Y 184.894,Z 578.49,A -85,B 0,C 180,E1 -22064.305,E2 -22064.305} C_VEL
LIN {X 0,Y 186.049,Z 573.517,A -85,B 0,C 180,E1 -22067.59,E2 -22067.59} C_VEL
LIN {X 0,Y 188.202,Z 566.883,A -85,B 0,C 180,E1 -22071.002,E2 -22071.002} C_VEL
LIN {X 0,Y 190.651,Z 559.682,A -85,B 0,C 180,E1 -22073.922,E2 -22073.922} C_VEL
LIN {X 0,Y 192.468,Z 551.798,A -85,B 0,C 180,E1 -22076.572,E2 -22076.572} C_VEL
LIN {X 0,Y 193.94,Z 543.189,A -85,B 0,C 180,E1 -22079.007,E2 -22079.007} C_VEL
LIN {X 0,Y 195.207,Z 532.863,A -85,B 0,C 180,E1 -22081.47,E2 -22081.47} C_VEL
LIN {X 0,Y 195.914,Z 521.228,A -85,B 0,C 180,E1 -22083.797,E2 -22083.797} C_VEL
LIN {X 0,Y 195.738,Z 508.973,A -85,B 0,C 180,E1 -22085.91,E2 -22085.91} C_VEL
LIN {X 0,Y 194.637,Z 495.9,A -85,B 0,C 180,E1 -22087.868,E2 -22087.868} C_VEL
LIN {X 0,Y 192.568,Z 483.204,A -85,B 0,C 180,E1 -22089.557,E2 -22089.557} C_VEL
LIN {X 0,Y 191.078,Z 476.99,A -85,B 0,C 180,E1 -22090.355,E2 -22090.355} C_VEL
LIN {X 0,Y 190.507,Z 474.249,A -85,B 0,C 180,E1 -22090.674,E2 -22090.674} C_VEL
LIN {X 0,Y 189.96,Z 470.311,A -85,B 0,C 180,E1 -22093.704,E2 -22093.704} C_VEL
LIN {X 0,Y 188.9,Z 464.95,A -85,B 0,C 180,E1 -22098.082,E2 -22098.082} C_VEL
LIN {X 0,Y 187.846,Z 459.035,A -85,B 0,C 180,E1 -22103.229,E2 -22103.229} C_VEL
LIN {X 0,Y 186.763,Z 453.841,A -85,B 0,C 180,E1 -22108.209,E2 -22108.209} C_VEL
LIN {X 0,Y 185.785,Z 449.326,A -85,B 0,C 180,E1 -22113.003,E2 -22113.003} C_VEL
LIN {X 0,Y 185.56,Z 448.369,A -85,B 0,C 180,E1 -22114.18,E2 -22114.18} C_VEL
LIN {X 0,Y 185.583,Z 448.361,A -85,B 0,C 180,E1 -22117.747,E2 -22117.747} C_VEL
LIN {X 0,Y 185.693,Z 448.356,A -85,B 0,C 180,E1 -22122.375,E2 -22122.375} C_VEL
LIN {X 0,Y 185.734,Z 448.354,A -85,B 0,C 180,E1 -22126.878,E2 -22126.878} C_VEL
LIN {X 0,Y 185.984,Z 448.32,A -85,B 0,C 180,E1 -22131.306,E2 -22131.306} C_VEL
LIN {X 0,Y 186.211,Z 448.291,A -85,B 0,C 180,E1 -22137.837,E2 -22137.837} C_VEL
LIN {X 0,Y 186.413,Z 448.263,A -85,B 0,C 180,E1 -22140,E2 -22140} C_VEL
LIN {X 0,Y 185.922,Z 448.325,A -85,B 0,C 180,E1 -22144.336,E2 -22144.336} C_VEL
LIN {X 0,Y 185.984,Z 448.318,A -85,B 0,C 180,E1 -22148.694,E2 -22148.694} C_VEL
LIN {X 0,Y 185.734,Z 448.312,A -85,B 0,C 180,E1 -22153.123,E2 -22153.123} C_VEL
LIN {X 0,Y 185.693,Z 448.308,A -85,B 0,C 180,E1 -22157.625,E2 -22157.625} C_VEL
LIN {X 0,Y 185.6,Z 448.362,A -85,B 0,C 180,E1 -22162.251,E2 -22162.251} C_VEL
LIN {X 0,Y 185.563,Z 448.323,A -85,B 0,C 180,E1 -22167.032,E2 -22167.032} C_VEL
LIN {X 0,Y 185.58,Z 448.33,A -85,B 0,C 180,E1 -22169.493,E2 -22169.493} C_VEL
LIN {X 0,Y 185.501,Z 448.371,A -85,B 0,C 180,E1 -22174.632,E2 -22174.632} C_VEL
LIN {X 0,Y 185.509,Z 448.377,A -85,B 0,C 180,E1 -22177.313,E2 -22177.313} C_VEL
LIN {X 0,Y 185.483,Z 448.376,A -85,B 0,C 180,E1 -22180.728,E2 -22180.728} C_VEL
LIN {X 0,Y 185.557,Z 448.37,A -85,B 0,C 180,E1 -22186.024,E2 -22186.024} C_VEL
LIN {X 0,Y 185.554,Z 448.367,A -85,B 0,C 180,E1 -22189.308,E2 -22189.308} C_VEL
LIN {X 0,Y 186.543,Z 451.168,A -85,B 0,C 180,E1 -22189.939,E2 -22189.939} C_VEL
LIN {X 0,Y 187.871,Z 452.828,A -85,B 0,C 180,E1 -22190.509,E2 -22190.509} C_VEL
LIN {X 0,Y 192.876,Z 462.773,A -85,B 0,C 180,E1 -22193.287,E2 -22193.287} C_VEL
LIN {X 0,Y 196.588,Z 471.534,A -85,B 0,C 180,E1 -22195.762,E2 -22195.762} C_VEL
LIN {X 0,Y 199.794,Z 481.033,A -85,B 0,C 180,E1 -22198.543,E2 -22198.543} C_VEL
LIN {X 0,Y 201.895,Z 490.133,A -85,B 0,C 180,E1 -22201.34,E2 -22201.34} C_VEL
LIN {X 0,Y 202.122,Z 493.135,A -85,B 0,C 180,E1 -22202.254,E2 -22202.254} C_VEL
LIN {X 0,Y 198.996,Z 502.899,A -85,B 0,C 180,E1 -22204.925,E2 -22204.925} C_VEL
LIN {X 0,Y 195.891,Z 511.389,A -85,B 0,C 180,E1 -22207.87,E2 -22207.87} C_VEL
LIN {X 0,Y 193.109,Z 518.571,A -85,B 0,C 180,E1 -22211.129,E2 -22211.129} C_VEL
LIN {X 0,Y 191.224,Z 523.495,A -85,B 0,C 180,E1 -22213.999,E2 -22213.999} C_VEL
LIN {X 0,Y 189.323,Z 527.733,A -85,B 0,C 180,E1 -22217.13,E2 -22217.13} C_VEL
LIN {X 0,Y 188.334,Z 529.966,A -85,B 0,C 180,E1 -22219.246,E2 -22219.246} C_VEL
LIN {X 0,Y 187.497,Z 531.786,A -85,B 0,C 180,E1 -22221.377,E2 -22221.377} C_VEL
LIN {X 0,Y 186.841,Z 533.154,A -85,B 0,C 180,E1 -22223.52,E2 -22223.52} C_VEL
LIN {X 0,Y 186.434,Z 534.675,A -85,B 0,C 180,E1 -22227.839,E2 -22227.839} C_VEL
LIN {X 0,Y 186.377,Z 534.894,A -85,B 0,C 180,E1 -22230,E2 -22230} C_VEL
LIN {X 0,Y 186.433,Z 534.707,A -85,B 0,C 180,E1 -22232.16,E2 -22232.16} C_VEL
LIN {X 0,Y 186.83,Z 533.228,A -85,B 0,C 180,E1 -22236.48,E2 -22236.48} C_VEL
LIN {X 0,Y 187.48,Z 531.894,A -85,B 0,C 180,E1 -22238.624,E2 -22238.624} C_VEL
LIN {X 0,Y 188.854,Z 529.067,A -85,B 0,C 180,E1 -22241.81,E2 -22241.81} C_VEL
LIN {X 0,Y 190.576,Z 525.245,A -85,B 0,C 180,E1 -22244.96,E2 -22244.96} C_VEL
LIN {X 0,Y 192.839,Z 519.323,A -85,B 0,C 180,E1 -22248.635,E2 -22248.635} C_VEL
LIN {X 0,Y 195.428,Z 512.922,A -85,B 0,C 180,E1 -22251.63,E2 -22251.63} C_VEL
LIN {X 0,Y 198.419,Z 504.878,A -85,B 0,C 180,E1 -22254.594,E2 -22254.594} C_VEL
LIN {X 0,Y 201.062,Z 496.644,A -85,B 0,C 180,E1 -22257.027,E2 -22257.027} C_VEL
LIN {X 0,Y 202.335,Z 492.323,A -85,B 0,C 180,E1 -22258.113,E2 -22258.113} C_VEL
LIN {X 0,Y 200.702,Z 484.494,A -85,B 0,C 180,E1 -22260.588,E2 -22260.588} C_VEL
LIN {X 0,Y 198.668,Z 477.294,A -85,B 0,C 180,E1 -22262.722,E2 -22262.722} C_VEL
LIN {X 0,Y 195.203,Z 468.016,A -85,B 0,C 180,E1 -22265.4,E2 -22265.4} C_VEL
LIN {X 0,Y 191.219,Z 459.377,A -85,B 0,C 180,E1 -22267.846,E2 -22267.846} C_VEL
LIN {X 0,Y 187.892,Z 452.786,A -85,B 0,C 180,E1 -22269.676,E2 -22269.676} C_VEL
LIN {X 0,Y 186.075,Z 450.207,A -85,B 0,C 180,E1 -22270.496,E2 -22270.496} C_VEL
LIN {X 0,Y 185.577,Z 448.369,A -85,B 0,C 180,E1 -22270.878,E2 -22270.878} C_VEL
LIN {X 0,Y 185.559,Z 448.369,A -85,B 0,C 180,E1 -22273.977,E2 -22273.977} C_VEL
LIN {X 0,Y 185.482,Z 448.376,A -85,B 0,C 180,E1 -22279.271,E2 -22279.271} C_VEL
LIN {X 0,Y 185.509,Z 448.372,A -85,B 0,C 180,E1 -22282.711,E2 -22282.711} C_VEL
LIN {X 0,Y 185.543,Z 448.366,A -85,B 0,C 180,E1 -22287.975,E2 -22287.975} C_VEL
LIN {X 0,Y 185.582,Z 448.369,A -85,B 0,C 180,E1 -22290.577,E2 -22290.577} C_VEL
LIN {X 0,Y 185.589,Z 448.367,A -85,B 0,C 180,E1 -22295.383,E2 -22295.383} C_VEL
LIN {X 0,Y 185.696,Z 448.351,A -85,B 0,C 180,E1 -22301.115,E2 -22301.115} C_VEL
LIN {X 0,Y 185.701,Z 448.351,A -85,B 0,C 180,E1 -22304.638,E2 -22304.638} C_VEL
LIN {X 0,Y 185.89,Z 448.326,A -85,B 0,C 180,E1 -22309.418,E2 -22309.418} C_VEL
LIN {X 0,Y 185.948,Z 448.311,A -85,B 0,C 180,E1 -22313.489,E2 -22313.489} C_VEL
LIN {X 0,Y 186.209,Z 448.288,A -85,B 0,C 180,E1 -22317.837,E2 -22317.837} C_VEL
LIN {X 0,Y 186.412,Z 448.259,A -85,B 0,C 180,E1 -22320,E2 -22320} C_VEL
LIN {X 0,Y 185.923,Z 448.325,A -85,B 0,C 180,E1 -22324.336,E2 -22324.336} C_VEL
LIN {X 0,Y 185.983,Z 448.31,A -85,B 0,C 180,E1 -22328.694,E2 -22328.694} C_VEL
LIN {X 0,Y 185.733,Z 448.341,A -85,B 0,C 180,E1 -22333.123,E2 -22333.123} C_VEL
LIN {X 0,Y 185.692,Z 448.349,A -85,B 0,C 180,E1 -22337.625,E2 -22337.625} C_VEL
LIN {X 0,Y 185.583,Z 448.371,A -85,B 0,C 180,E1 -22342.253,E2 -22342.253} C_VEL
LIN {X 0,Y 185.567,Z 448.405,A -85,B 0,C 180,E1 -22345.819,E2 -22345.819} C_VEL
LIN {X 0,Y 186.389,Z 452.077,A -85,B 0,C 180,E1 -22349.86,E2 -22349.86} C_VEL
LIN {X 0,Y 187.357,Z 456.624,A -85,B 0,C 180,E1 -22354.386,E2 -22354.386} C_VEL
LIN {X 0,Y 188.387,Z 462.068,A -85,B 0,C 180,E1 -22359.361,E2 -22359.361} C_VEL
LIN {X 0,Y 189.586,Z 468.523,A -85,B 0,C 180,E1 -22364.776,E2 -22364.776} C_VEL
LIN {X 0,Y 190.477,Z 473.606,A -85,B 0,C 180,E1 -22368.775,E2 -22368.775} C_VEL
LIN {X 0,Y 190.498,Z 474.275,A -85,B 0,C 180,E1 -22369.263,E2 -22369.263} C_VEL
LIN {X 0,Y 191.508,Z 478.175,A -85,B 0,C 180,E1 -22369.741,E2 -22369.741} C_VEL
LIN {X 0,Y 194.14,Z 491.715,A -85,B 0,C 180,E1 -22371.501,E2 -22371.501} C_VEL
LIN {X 0,Y 195.606,Z 505.157,A -85,B 0,C 180,E1 -22373.434,E2 -22373.434} C_VEL
LIN {X 0,Y 196.011,Z 516.684,A -85,B 0,C 180,E1 -22375.32,E2 -22375.32} C_VEL
LIN {X 0,Y 195.676,Z 527.757,A -85,B 0,C 180,E1 -22377.402,E2 -22377.402} C_VEL
LIN {X 0,Y 194.611,Z 539.038,A -85,B 0,C 180,E1 -22379.905,E2 -22379.905} C_VEL
LIN {X 0,Y 193.124,Z 548.373,A -85,B 0,C 180,E1 -22382.355,E2 -22382.355} C_VEL
LIN {X 0,Y 191.443,Z 556.87,A -85,B 0,C 180,E1 -22385.028,E2 -22385.028} C_VEL
LIN {X 0,Y 189.3,Z 563.843,A -85,B 0,C 180,E1 -22387.633,E2 -22387.633} C_VEL
LIN {X 0,Y 186.948,Z 570.696,A -85,B 0,C 180,E1 -22390.796,E2 -22390.796} C_VEL
LIN {X 0,Y 185.222,Z 577.058,A -85,B 0,C 180,E1 -22394.597,E2 -22394.597} C_VEL
LIN {X 0,Y 184.455,Z 581.257,A -85,B 0,C 180,E1 -22397.904,E2 -22397.904} C_VEL
LIN {X 0,Y 184.386,Z 585.221,A -85,B 0,C 180,E1 -22402.311,E2 -22402.311} C_VEL
LIN {X 0,Y 184.862,Z 587.103,A -85,B 0,C 180,E1 -22405.639,E2 -22405.639} C_VEL
LIN {X 0,Y 185.831,Z 588.128,A -85,B 0,C 180,E1 -22410,E2 -22410} C_VEL
LIN {X 0,Y 184.852,Z 587.083,A -85,B 0,C 180,E1 -22414.361,E2 -22414.361} C_VEL
LIN {X 0,Y 184.375,Z 585.211,A -85,B 0,C 180,E1 -22417.652,E2 -22417.652} C_VEL
LIN {X 0,Y 183.662,Z 583.817,A -85,B 0,C 180,E1 -22419.425,E2 -22419.425} C_VEL
LIN {X 0,Y 180.994,Z 580.83,A -85,B 0,C 180,E1 -22422.279,E2 -22422.279} C_VEL
LIN {X 0,Y 178.709,Z 577.162,A -85,B 0,C 180,E1 -22425.138,E2 -22425.138} C_VEL
LIN {X 0,Y 178.619,Z 574.693,A -85,B 0,C 180,E1 -22426.869,E2 -22426.869} C_VEL
LIN {X 0,Y 180.498,Z 568.507,A -85,B 0,C 180,E1 -22430.514,E2 -22430.514} C_VEL
LIN {X 0,Y 183.152,Z 561.413,A -85,B 0,C 180,E1 -22433.761,E2 -22433.761} C_VEL
LIN {X 0,Y 185.205,Z 554.108,A -85,B 0,C 180,E1 -22436.48,E2 -22436.48} C_VEL
LIN {X 0,Y 186.991,Z 545.234,A -85,B 0,C 180,E1 -22439.249,E2 -22439.249} C_VEL
LIN {X 0,Y 188.41,Z 535.478,A -85,B 0,C 180,E1 -22441.796,E2 -22441.796} C_VEL
LIN {X 0,Y 189.364,Z 524.828,A -85,B 0,C 180,E1 -22444.153,E2 -22444.153} C_VEL
LIN {X 0,Y 189.622,Z 513.202,A -85,B 0,C 180,E1 -22446.371,E2 -22446.371} C_VEL
LIN {X 0,Y 189.007,Z 500.759,A -85,B 0,C 180,E1 -22448.447,E2 -22448.447} C_VEL
LIN {X 0,Y 187.395,Z 487.795,A -85,B 0,C 180,E1 -22450.362,E2 -22450.362} C_VEL
LIN {X 0,Y 185.373,Z 478.216,A -85,B 0,C 180,E1 -22451.701,E2 -22451.701} C_VEL
LIN {X 0,Y 183.603,Z 474.432,A -85,B 0,C 180,E1 -22452.434,E2 -22452.434} C_VEL
LIN {X 0,Y 183.212,Z 472.849,A -85,B 0,C 180,E1 -22452.707,E2 -22452.707} C_VEL
LIN {X 0,Y 181.982,Z 466.518,A -85,B 0,C 180,E1 -22458.029,E2 -22458.029} C_VEL
LIN {X 0,Y 181,Z 461.024,A -85,B 0,C 180,E1 -22462.998,E2 -22462.998} C_VEL
LIN {X 0,Y 179.935,Z 455.785,A -85,B 0,C 180,E1 -22468.179,E2 -22468.179} C_VEL
LIN {X 0,Y 178.958,Z 451.268,A -85,B 0,C 180,E1 -22473.152,E2 -22473.152} C_VEL
LIN {X 0,Y 178.541,Z 449.246,A -85,B 0,C 180,E1 -22475.805,E2 -22475.805} C_VEL
LIN {X 0,Y 178.652,Z 449.233,A -85,B 0,C 180,E1 -22481.657,E2 -22481.657} C_VEL
LIN {X 0,Y 178.662,Z 449.235,A -85,B 0,C 180,E1 -22486.348,E2 -22486.348} C_VEL
LIN {X 0,Y 178.913,Z 449.2,A -85,B 0,C 180,E1 -22490.96,E2 -22490.96} C_VEL
LIN {X 0,Y 179.156,Z 449.169,A -85,B 0,C 180,E1 -22497.752,E2 -22497.752} C_VEL
LIN {X 0,Y 179.376,Z 449.139,A -85,B 0,C 180,E1 -22500,E2 -22500} C_VEL
LIN {X 0,Y 178.87,Z 449.203,A -85,B 0,C 180,E1 -22504.507,E2 -22504.507} C_VEL
LIN {X 0,Y 178.913,Z 449.199,A -85,B 0,C 180,E1 -22509.04,E2 -22509.04} C_VEL
LIN {X 0,Y 178.661,Z 449.182,A -85,B 0,C 180,E1 -22513.652,E2 -22513.652} C_VEL
LIN {X 0,Y 178.626,Z 449.21,A -85,B 0,C 180,E1 -22519.216,E2 -22519.216} C_VEL
LIN {X 0,Y 178.537,Z 449.217,A -85,B 0,C 180,E1 -22525.124,E2 -22525.124} C_VEL
LIN {X 0,Y 178.479,Z 449.232,A -85,B 0,C 180,E1 -22530.791,E2 -22530.791} C_VEL
LIN {X 0,Y 178.486,Z 449.247,A -85,B 0,C 180,E1 -22534.219,E2 -22534.219} C_VEL
LIN {X 0,Y 178.403,Z 449.257,A -85,B 0,C 180,E1 -22539.073,E2 -22539.073} C_VEL
LIN {X 0,Y 178.422,Z 449.26,A -85,B 0,C 180,E1 -22542.038,E2 -22542.038} C_VEL
LIN {X 0,Y 178.516,Z 449.24,A -85,B 0,C 180,E1 -22547.265,E2 -22547.265} C_VEL
LIN {X 0,Y 179.522,Z 452.139,A -85,B 0,C 180,E1 -22547.98,E2 -22547.98} C_VEL
LIN {X 0,Y 181.02,Z 454.126,A -85,B 0,C 180,E1 -22548.698,E2 -22548.698} C_VEL
LIN {X 0,Y 186.22,Z 464.134,A -85,B 0,C 180,E1 -22551.772,E2 -22551.772} C_VEL
LIN {X 0,Y 190.035,Z 472.893,A -85,B 0,C 180,E1 -22554.451,E2 -22554.451} C_VEL
LIN {X 0,Y 193.138,Z 482.047,A -85,B 0,C 180,E1 -22557.298,E2 -22557.298} C_VEL
LIN {X 0,Y 195.011,Z 490.083,A -85,B 0,C 180,E1 -22559.876,E2 -22559.876} C_VEL
LIN {X 0,Y 195.795,Z 494.51,A -85,B 0,C 180,E1 -22561.387,E2 -22561.387} C_VEL
LIN {X 0,Y 192.655,Z 503.907,A -85,B 0,C 180,E1 -22564.039,E2 -22564.039} C_VEL
LIN {X 0,Y 189.4,Z 512.396,A -85,B 0,C 180,E1 -22567.069,E2 -22567.069} C_VEL
LIN {X 0,Y 186.473,Z 519.578,A -85,B 0,C 180,E1 -22570.43,E2 -22570.43} C_VEL
LIN {X 0,Y 184.48,Z 524.501,A -85,B 0,C 180,E1 -22573.398,E2 -22573.398} C_VEL
LIN {X 0,Y 182.479,Z 528.739,A -85,B 0,C 180,E1 -22576.639,E2 -22576.639} C_VEL
LIN {X 0,Y 181.434,Z 530.972,A -85,B 0,C 180,E1 -22578.832,E2 -22578.832} C_VEL
LIN {X 0,Y 180.552,Z 532.792,A -85,B 0,C 180,E1 -22581.042,E2 -22581.042} C_VEL
LIN {X 0,Y 179.859,Z 534.16,A -85,B 0,C 180,E1 -22583.268,E2 -22583.268} C_VEL
LIN {X 0,Y 179.412,Z 535.68,A -85,B 0,C 180,E1 -22587.755,E2 -22587.755} C_VEL
LIN {X 0,Y 179.35,Z 535.899,A -85,B 0,C 180,E1 -22590,E2 -22590} C_VEL
LIN {X 0,Y 179.411,Z 535.712,A -85,B 0,C 180,E1 -22592.245,E2 -22592.245} C_VEL
LIN {X 0,Y 179.849,Z 534.233,A -85,B 0,C 180,E1 -22596.732,E2 -22596.732} C_VEL
LIN {X 0,Y 180.534,Z 532.898,A -85,B 0,C 180,E1 -22598.958,E2 -22598.958} C_VEL
LIN {X 0,Y 181.98,Z 530.072,A -85,B 0,C 180,E1 -22602.263,E2 -22602.263} C_VEL
LIN {X 0,Y 183.795,Z 526.249,A -85,B 0,C 180,E1 -22605.525,E2 -22605.525} C_VEL
LIN {X 0,Y 186.191,Z 520.329,A -85,B 0,C 180,E1 -22609.324,E2 -22609.324} C_VEL
LIN {X 0,Y 188.913,Z 513.926,A -85,B 0,C 180,E1 -22612.416,E2 -22612.416} C_VEL
LIN {X 0,Y 192.051,Z 505.881,A -85,B 0,C 180,E1 -22615.466,E2 -22615.466} C_VEL
LIN {X 0,Y 194.835,Z 497.645,A -85,B 0,C 180,E1 -22617.965,E2 -22617.965} C_VEL
LIN {X 0,Y 195.714,Z 494.888,A -85,B 0,C 180,E1 -22618.674,E2 -22618.674} C_VEL
LIN {X 0,Y 195.097,Z 490.042,A -85,B 0,C 180,E1 -22620.286,E2 -22620.286} C_VEL
LIN {X 0,Y 192.96,Z 481.324,A -85,B 0,C 180,E1 -22623.101,E2 -22623.101} C_VEL
LIN {X 0,Y 189.804,Z 472.325,A -85,B 0,C 180,E1 -22625.906,E2 -22625.906} C_VEL
LIN {X 0,Y 186.116,Z 463.818,A -85,B 0,C 180,E1 -22628.5,E2 -22628.5} C_VEL
LIN {X 0,Y 182.582,Z 457.015,A -85,B 0,C 180,E1 -22630.601,E2 -22630.601} C_VEL
LIN {X 0,Y 180.493,Z 453.329,A -85,B 0,C 180,E1 -22631.763,E2 -22631.763} C_VEL
LIN {X 0,Y 178.88,Z 450.803,A -85,B 0,C 180,E1 -22632.594,E2 -22632.594} C_VEL
LIN {X 0,Y 178.527,Z 449.249,A -85,B 0,C 180,E1 -22632.996,E2 -22632.996} C_VEL
LIN {X 0,Y 178.419,Z 449.255,A -85,B 0,C 180,E1 -22638.454,E2 -22638.454} C_VEL
LIN {X 0,Y 178.424,Z 449.255,A -85,B 0,C 180,E1 -22643.783,E2 -22643.783} C_VEL
LIN {X 0,Y 178.487,Z 449.248,A -85,B 0,C 180,E1 -22646.546,E2 -22646.546} C_VEL
LIN {X 0,Y 178.523,Z 449.248,A -85,B 0,C 180,E1 -22650.007,E2 -22650.007} C_VEL
LIN {X 0,Y 178.536,Z 449.248,A -85,B 0,C 180,E1 -22654.876,E2 -22654.876} C_VEL
LIN {X 0,Y 178.64,Z 449.232,A -85,B 0,C 180,E1 -22660.769,E2 -22660.769} C_VEL
LIN {X 0,Y 178.662,Z 449.229,A -85,B 0,C 180,E1 -22666.348,E2 -22666.348} C_VEL
LIN {X 0,Y 178.912,Z 449.199,A -85,B 0,C 180,E1 -22670.96,E2 -22670.96} C_VEL
LIN {X 0,Y 179.154,Z 449.167,A -85,B 0,C 180,E1 -22677.752,E2 -22677.752} C_VEL
LIN {X 0,Y 179.374,Z 449.135,A -85,B 0,C 180,E1 -22680,E2 -22680} C_VEL
LIN {X 0,Y 178.871,Z 449.204,A -85,B 0,C 180,E1 -22684.507,E2 -22684.507} C_VEL
LIN {X 0,Y 178.912,Z 449.192,A -85,B 0,C 180,E1 -22689.04,E2 -22689.04} C_VEL
LIN {X 0,Y 178.661,Z 449.224,A -85,B 0,C 180,E1 -22693.652,E2 -22693.652} C_VEL
LIN {X 0,Y 178.623,Z 449.236,A -85,B 0,C 180,E1 -22699.215,E2 -22699.215} C_VEL
LIN {X 0,Y 178.566,Z 449.413,A -85,B 0,C 180,E1 -22704.533,E2 -22704.533} C_VEL
LIN {X 0,Y 179.469,Z 453.535,A -85,B 0,C 180,E1 -22709.308,E2 -22709.308} C_VEL
LIN {X 0,Y 180.419,Z 458.195,A -85,B 0,C 180,E1 -22714.162,E2 -22714.162} C_VEL
LIN {X 0,Y 181.444,Z 463.532,A -85,B 0,C 180,E1 -22719.225,E2 -22719.225} C_VEL
LIN {X 0,Y 182.708,Z 470.247,A -85,B 0,C 180,E1 -22725.076,E2 -22725.076} C_VEL
LIN {X 0,Y 183.239,Z 473,A -85,B 0,C 180,E1 -22727.284,E2 -22727.284} C_VEL
LIN {X 0,Y 184.523,Z 476.633,A -85,B 0,C 180,E1 -22727.861,E2 -22727.861} C_VEL
LIN {X 0,Y 185.466,Z 478.602,A -85,B 0,C 180,E1 -22728.262,E2 -22728.262} C_VEL
LIN {X 0,Y 187.168,Z 486.266,A -85,B 0,C 180,E1 -22729.352,E2 -22729.352} C_VEL
LIN {X 0,Y 188.892,Z 498.69,A -85,B 0,C 180,E1 -22731.17,E2 -22731.17} C_VEL
LIN {X 0,Y 189.652,Z 510.269,A -85,B 0,C 180,E1 -22733.051,E2 -22733.051} C_VEL
LIN {X 0,Y 189.571,Z 522.028,A -85,B 0,C 180,E1 -22735.214,E2 -22735.214} C_VEL
LIN {X 0,Y 188.754,Z 533.306,A -85,B 0,C 180,E1 -22737.64,E2 -22737.64} C_VEL
LIN {X 0,Y 187.408,Z 542.909,A -85,B 0,C 180,E1 -22740.05,E2 -22740.05} C_VEL
LIN {X 0,Y 185.62,Z 552.636,A -85,B 0,C 180,E1 -22742.977,E2 -22742.977} C_VEL
LIN {X 0,Y 183.628,Z 560.198,A -85,B 0,C 180,E1 -22745.705,E2 -22745.705} C_VEL
LIN {X 0,Y 180.827,Z 567.852,A -85,B 0,C 180,E1 -22749.085,E2 -22749.085} C_VEL
LIN {X 0,Y 178.748,Z 574.366,A -85,B 0,C 180,E1 -22752.85,E2 -22752.85} C_VEL
LIN {X 0,Y 177.681,Z 578.932,A -85,B 0,C 180,E1 -22756.271,E2 -22756.271} C_VEL
LIN {X 0,Y 177.254,Z 582.433,A -85,B 0,C 180,E1 -22759.722,E2 -22759.722} C_VEL
LIN {X 0,Y 177.409,Z 584.948,A -85,B 0,C 180,E1 -22763.175,E2 -22763.175} C_VEL
LIN {X 0,Y 177.767,Z 586.086,A -85,B 0,C 180,E1 -22765.465,E2 -22765.465} C_VEL
LIN {X 0,Y 178.785,Z 587.12,A -85,B 0,C 180,E1 -22770,E2 -22770} C_VEL
LIN {X 0,Y 177.756,Z 586.064,A -85,B 0,C 180,E1 -22774.536,E2 -22774.536} C_VEL
LIN {X 0,Y 177.317,Z 584.342,A -85,B 0,C 180,E1 -22777.743,E2 -22777.743} C_VEL
LIN {X 0,Y 177.328,Z 581.33,A -85,B 0,C 180,E1 -22781.43,E2 -22781.43} C_VEL
LIN {X 0,Y 177.941,Z 577.461,A -85,B 0,C 180,E1 -22784.876,E2 -22784.876} C_VEL
LIN {X 0,Y 178.619,Z 574.693,A -85,B 0,C 180,E1 -22786.869,E2 -22786.869} C_VEL
LIN {X 0,Y 178.745,Z 572.062,A -85,B 0,C 180,E1 -22788.565,E2 -22788.565} C_VEL
LIN {X 0,Y 177.609,Z 567.253,A -85,B 0,C 180,E1 -22791.329,E2 -22791.329} C_VEL
LIN {X 0,Y 176.752,Z 561.866,A -85,B 0,C 180,E1 -22794.012,E2 -22794.012} C_VEL
LIN {X 0,Y 177.305,Z 558.308,A -85,B 0,C 180,E1 -22795.537,E2 -22795.537} C_VEL
LIN {X 0,Y 179.437,Z 549.69,A -85,B 0,C 180,E1 -22798.672,E2 -22798.672} C_VEL
LIN {X 0,Y 181.187,Z 540.577,A -85,B 0,C 180,E1 -22801.422,E2 -22801.422} C_VEL
LIN {X 0,Y 182.503,Z 530.697,A -85,B 0,C 180,E1 -22803.944,E2 -22803.944} C_VEL
LIN {X 0,Y 183.331,Z 519.441,A -85,B 0,C 180,E1 -22806.386,E2 -22806.386} C_VEL
LIN {X 0,Y 183.292,Z 506.758,A -85,B 0,C 180,E1 -22808.774,E2 -22808.774} C_VEL
LIN {X 0,Y 182.234,Z 493.586,A -85,B 0,C 180,E1 -22810.967,E2 -22810.967} C_VEL
LIN {X 0,Y 180.566,Z 483.349,A -85,B 0,C 180,E1 -22812.543,E2 -22812.543} C_VEL
LIN {X 0,Y 179.5,Z 480.352,A -85,B 0,C 180,E1 -22813.123,E2 -22813.123} C_VEL
LIN {X 0,Y 178.122,Z 476.915,A -85,B 0,C 180,E1 -22813.804,E2 -22813.804} C_VEL
LIN {X 0,Y 176.17,Z 473.132,A -85,B 0,C 180,E1 -22814.673,E2 -22814.673} C_VEL
LIN {X 0,Y 175.718,Z 471.492,A -85,B 0,C 180,E1 -22814.929,E2 -22814.929} C_VEL
LIN {X 0,Y 174.671,Z 465.918,A -85,B 0,C 180,E1 -22819.926,E2 -22819.926} C_VEL
LIN {X 0,Y 173.927,Z 461.77,A -85,B 0,C 180,E1 -22823.917,E2 -22823.917} C_VEL
LIN {X 0,Y 173.038,Z 457.367,A -85,B 0,C 180,E1 -22828.532,E2 -22828.532} C_VEL
LIN {X 0,Y 172.146,Z 453.201,A -85,B 0,C 180,E1 -22833.315,E2 -22833.315} C_VEL
LIN {X 0,Y 171.461,Z 450.12,A -85,B 0,C 180,E1 -22837.401,E2 -22837.401} C_VEL
LIN {X 0,Y 171.581,Z 450.112,A -85,B 0,C 180,E1 -22840.872,E2 -22840.872} C_VEL
LIN {X 0,Y 171.579,Z 450.115,A -85,B 0,C 180,E1 -22845.773,E2 -22845.773} C_VEL
LIN {X 0,Y 171.85,Z 450.08,A -85,B 0,C 180,E1 -22850.585,E2 -22850.585} C_VEL
LIN {X 0,Y 171.82,Z 450.086,A -85,B 0,C 180,E1 -22855.308,E2 -22855.308} C_VEL
LIN {X 0,Y 172.338,Z 450.016,A -85,B 0,C 180,E1 -22860,E2 -22860} C_VEL
LIN {X 0,Y 171.818,Z 450.082,A -85,B 0,C 180,E1 -22864.693,E2 -22864.693} C_VEL
LIN {X 0,Y 171.85,Z 450.078,A -85,B 0,C 180,E1 -22869.415,E2 -22869.415} C_VEL
LIN {X 0,Y 171.578,Z 450.054,A -85,B 0,C 180,E1 -22874.227,E2 -22874.227} C_VEL
LIN {X 0,Y 171.547,Z 450.096,A -85,B 0,C 180,E1 -22879.562,E2 -22879.562} C_VEL
LIN {X 0,Y 171.471,Z 450.087,A -85,B 0,C 180,E1 -22885.616,E2 -22885.616} C_VEL
LIN {X 0,Y 171.442,Z 450.103,A -85,B 0,C 180,E1 -22890.585,E2 -22890.585} C_VEL
LIN {X 0,Y 171.395,Z 450.126,A -85,B 0,C 180,E1 -22895.035,E2 -22895.035} C_VEL
LIN {X 0,Y 171.363,Z 450.135,A -85,B 0,C 180,E1 -22898.809,E2 -22898.809} C_VEL
LIN {X 0,Y 171.431,Z 450.128,A -85,B 0,C 180,E1 -22904.955,E2 -22904.955} C_VEL
LIN {X 0,Y 172.447,Z 453.003,A -85,B 0,C 180,E1 -22905.751,E2 -22905.751} C_VEL
LIN {X 0,Y 174.098,Z 455.066,A -85,B 0,C 180,E1 -22906.605,E2 -22906.605} C_VEL
LIN {X 0,Y 179.306,Z 464.791,A -85,B 0,C 180,E1 -22909.889,E2 -22909.889} C_VEL
LIN {X 0,Y 183.458,Z 474.098,A -85,B 0,C 180,E1 -22912.977,E2 -22912.977} C_VEL
LIN {X 0,Y 186.06,Z 481.734,A -85,B 0,C 180,E1 -22915.487,E2 -22915.487} C_VEL
LIN {X 0,Y 188.171,Z 489.545,A -85,B 0,C 180,E1 -22918.159,E2 -22918.159} C_VEL
LIN {X 0,Y 189.287,Z 495.916,A -85,B 0,C 180,E1 -22920.421,E2 -22920.421} C_VEL
LIN {X 0,Y 188.795,Z 498.13,A -85,B 0,C 180,E1 -22921.057,E2 -22921.057} C_VEL
LIN {X 0,Y 185.784,Z 506.486,A -85,B 0,C 180,E1 -22923.609,E2 -22923.609} C_VEL
LIN {X 0,Y 182.442,Z 514.606,A -85,B 0,C 180,E1 -22926.743,E2 -22926.743} C_VEL
LIN {X 0,Y 179.846,Z 520.618,A -85,B 0,C 180,E1 -22929.698,E2 -22929.698} C_VEL
LIN {X 0,Y 177.757,Z 525.508,A -85,B 0,C 180,E1 -22932.751,E2 -22932.751} C_VEL
LIN {X 0,Y 175.649,Z 529.745,A -85,B 0,C 180,E1 -22936.109,E2 -22936.109} C_VEL
LIN {X 0,Y 174.545,Z 531.978,A -85,B 0,C 180,E1 -22938.385,E2 -22938.385} C_VEL
LIN {X 0,Y 173.613,Z 533.798,A -85,B 0,C 180,E1 -22940.681,E2 -22940.681} C_VEL
LIN {X 0,Y 172.882,Z 535.165,A -85,B 0,C 180,E1 -22942.995,E2 -22942.995} C_VEL
LIN {X 0,Y 172.39,Z 536.685,A -85,B 0,C 180,E1 -22947.663,E2 -22947.663} C_VEL
LIN {X 0,Y 172.323,Z 536.904,A -85,B 0,C 180,E1 -22950,E2 -22950} C_VEL
LIN {X 0,Y 172.389,Z 536.717,A -85,B 0,C 180,E1 -22952.336,E2 -22952.336} C_VEL
LIN {X 0,Y 172.871,Z 535.237,A -85,B 0,C 180,E1 -22957.005,E2 -22957.005} C_VEL
LIN {X 0,Y 173.595,Z 533.903,A -85,B 0,C 180,E1 -22959.319,E2 -22959.319} C_VEL
LIN {X 0,Y 175.119,Z 531.076,A -85,B 0,C 180,E1 -22962.752,E2 -22962.752} C_VEL
LIN {X 0,Y 177.034,Z 527.253,A -85,B 0,C 180,E1 -22966.134,E2 -22966.134} C_VEL
LIN {X 0,Y 179.582,Z 521.318,A -85,B 0,C 180,E1 -22970.074,E2 -22970.074} C_VEL
LIN {X 0,Y 182.937,Z 513.729,A -85,B 0,C 180,E1 -22973.79,E2 -22973.79} C_VEL
LIN {X 0,Y 186.296,Z 505.351,A -85,B 0,C 180,E1 -22976.917,E2 -22976.917} C_VEL
LIN {X 0,Y 189.311,Z 496.293,A -85,B 0,C 180,E1 -22979.618,E2 -22979.618} C_VEL
LIN {X 0,Y 188.034,Z 488.768,A -85,B 0,C 180,E1 -22982.273,E2 -22982.273} C_VEL
LIN {X 0,Y 185.7,Z 480.468,A -85,B 0,C 180,E1 -22985.098,E2 -22985.098} C_VEL
LIN {X 0,Y 182.41,Z 471.486,A -85,B 0,C 180,E1 -22988.058,E2 -22988.058} C_VEL
LIN {X 0,Y 178.305,Z 462.706,A -85,B 0,C 180,E1 -22990.98,E2 -22990.98} C_VEL
LIN {X 0,Y 174.302,Z 455.515,A -85,B 0,C 180,E1 -22993.466,E2 -22993.466} C_VEL
LIN {X 0,Y 171.811,Z 451.725,A -85,B 0,C 180,E1 -22994.866,E2 -22994.866} C_VEL
LIN {X 0,Y 171.405,Z 450.129,A -85,B 0,C 180,E1 -22995.272,E2 -22995.272} C_VEL
LIN {X 0,Y 171.363,Z 450.141,A -85,B 0,C 180,E1 -23001.191,E2 -23001.191} C_VEL
LIN {X 0,Y 171.399,Z 450.137,A -85,B 0,C 180,E1 -23005.092,E2 -23005.092} C_VEL
LIN {X 0,Y 171.449,Z 450.129,A -85,B 0,C 180,E1 -23010.534,E2 -23010.534} C_VEL
LIN {X 0,Y 171.46,Z 450.127,A -85,B 0,C 180,E1 -23015.802,E2 -23015.802} C_VEL
LIN {X 0,Y 171.597,Z 450.109,A -85,B 0,C 180,E1 -23020.873,E2 -23020.873} C_VEL
LIN {X 0,Y 171.582,Z 450.112,A -85,B 0,C 180,E1 -23025.773,E2 -23025.773} C_VEL
LIN {X 0,Y 171.849,Z 450.079,A -85,B 0,C 180,E1 -23030.585,E2 -23030.585} C_VEL
LIN {X 0,Y 171.816,Z 450.064,A -85,B 0,C 180,E1 -23035.307,E2 -23035.307} C_VEL
LIN {X 0,Y 172.337,Z 450.011,A -85,B 0,C 180,E1 -23040,E2 -23040} C_VEL
LIN {X 0,Y 171.819,Z 450.084,A -85,B 0,C 180,E1 -23044.692,E2 -23044.692} C_VEL
LIN {X 0,Y 171.848,Z 450.075,A -85,B 0,C 180,E1 -23049.415,E2 -23049.415} C_VEL
LIN {X 0,Y 171.579,Z 450.109,A -85,B 0,C 180,E1 -23054.227,E2 -23054.227} C_VEL
LIN {X 0,Y 171.543,Z 450.117,A -85,B 0,C 180,E1 -23059.559,E2 -23059.559} C_VEL
LIN {X 0,Y 171.465,Z 450.276,A -85,B 0,C 180,E1 -23062.916,E2 -23062.916} C_VEL
LIN {X 0,Y 172.429,Z 454.345,A -85,B 0,C 180,E1 -23067.952,E2 -23067.952} C_VEL
LIN {X 0,Y 173.427,Z 459.013,A -85,B 0,C 180,E1 -23073.167,E2 -23073.167} C_VEL
LIN {X 0,Y 174.426,Z 464.518,A -85,B 0,C 180,E1 -23078.648,E2 -23078.648} C_VEL
LIN {X 0,Y 175.431,Z 470.198,A -85,B 0,C 180,E1 -23083.854,E2 -23083.854} C_VEL
LIN {X 0,Y 175.739,Z 471.611,A -85,B 0,C 180,E1 -23084.988,E2 -23084.988} C_VEL
LIN {X 0,Y 177.111,Z 475.255,A -85,B 0,C 180,E1 -23085.656,E2 -23085.656} C_VEL
LIN {X 0,Y 178.65,Z 478.02,A -85,B 0,C 180,E1 -23086.342,E2 -23086.342} C_VEL
LIN {X 0,Y 180.678,Z 483.648,A -85,B 0,C 180,E1 -23087.422,E2 -23087.422} C_VEL
LIN {X 0,Y 182.412,Z 494.295,A -85,B 0,C 180,E1 -23089.082,E2 -23089.082} C_VEL
LIN {X 0,Y 183.366,Z 506.923,A -85,B 0,C 180,E1 -23091.186,E2 -23091.186} C_VEL
LIN {X 0,Y 183.403,Z 519.605,A -85,B 0,C 180,E1 -23093.583,E2 -23093.583} C_VEL
LIN {X 0,Y 182.564,Z 530.996,A -85,B 0,C 180,E1 -23096.069,E2 -23096.069} C_VEL
LIN {X 0,Y 181.255,Z 540.661,A -85,B 0,C 180,E1 -23098.543,E2 -23098.543} C_VEL
LIN {X 0,Y 179.404,Z 549.874,A -85,B 0,C 180,E1 -23101.322,E2 -23101.322} C_VEL
LIN {X 0,Y 177.539,Z 557.768,A -85,B 0,C 180,E1 -23104.187,E2 -23104.187} C_VEL
LIN {X 0,Y 175.087,Z 564.572,A -85,B 0,C 180,E1 -23107.131,E2 -23107.131} C_VEL
LIN {X 0,Y 172.446,Z 571.569,A -85,B 0,C 180,E1 -23110.972,E2 -23110.972} C_VEL
LIN {X 0,Y 171.027,Z 576.517,A -85,B 0,C 180,E1 -23114.508,E2 -23114.508} C_VEL
LIN {X 0,Y 170.288,Z 580.357,A -85,B 0,C 180,E1 -23118.091,E2 -23118.091} C_VEL
LIN {X 0,Y 170.277,Z 583.49,A -85,B 0,C 180,E1 -23122.128,E2 -23122.128} C_VEL
LIN {X 0,Y 170.676,Z 585.068,A -85,B 0,C 180,E1 -23125.276,E2 -23125.276} C_VEL
LIN {X 0,Y 171.737,Z 586.112,A -85,B 0,C 180,E1 -23130,E2 -23130} C_VEL
LIN {X 0,Y 170.665,Z 585.047,A -85,B 0,C 180,E1 -23134.724,E2 -23134.724} C_VEL
LIN {X 0,Y 170.268,Z 583.467,A -85,B 0,C 180,E1 -23137.85,E2 -23137.85} C_VEL
LIN {X 0,Y 170.288,Z 580.301,A -85,B 0,C 180,E1 -23141.909,E2 -23141.909} C_VEL
LIN {X 0,Y 171.021,Z 576.435,A -85,B 0,C 180,E1 -23145.493,E2 -23145.493} C_VEL
LIN {X 0,Y 172.421,Z 571.461,A -85,B 0,C 180,E1 -23149.032,E2 -23149.032} C_VEL
LIN {X 0,Y 175.079,Z 564.457,A -85,B 0,C 180,E1 -23152.864,E2 -23152.864} C_VEL
LIN {X 0,Y 177.305,Z 558.308,A -85,B 0,C 180,E1 -23155.537,E2 -23155.537} C_VEL
LIN {X 0,Y 177.742,Z 554.639,A -85,B 0,C 180,E1 -23157.02,E2 -23157.02} C_VEL
LIN {X 0,Y 177.154,Z 550.964,A -85,B 0,C 180,E1 -23158.519,E2 -23158.519} C_VEL
LIN {X 0,Y 175.042,Z 541.904,A -85,B 0,C 180,E1 -23161.926,E2 -23161.926} C_VEL
LIN {X 0,Y 175.179,Z 537.519,A -85,B 0,C 180,E1 -23163.252,E2 -23163.252} C_VEL
LIN {X 0,Y 176.702,Z 525.555,A -85,B 0,C 180,E1 -23166.273,E2 -23166.273} C_VEL
LIN {X 0,Y 177.267,Z 514.333,A -85,B 0,C 180,E1 -23168.706,E2 -23168.706} C_VEL
LIN {X 0,Y 177.017,Z 502.056,A -85,B 0,C 180,E1 -23171.032,E2 -23171.032} C_VEL
LIN {X 0,Y 175.795,Z 489.482,A -85,B 0,C 180,E1 -23173.179,E2 -23173.179} C_VEL
LIN {X 0,Y 174.886,Z 485.164,A -85,B 0,C 180,E1 -23173.962,E2 -23173.962} C_VEL
LIN {X 0,Y 173.18,Z 480.963,A -85,B 0,C 180,E1 -23174.926,E2 -23174.926} C_VEL
LIN {X 0,Y 171.291,Z 476.569,A -85,B 0,C 180,E1 -23175.942,E2 -23175.942} C_VEL
LIN {X 0,Y 168.861,Z 472.172,A -85,B 0,C 180,E1 -23177.139,E2 -23177.139} C_VEL
LIN {X 0,Y 168.172,Z 469.87,A -85,B 0,C 180,E1 -23177.633,E2 -23177.633} C_VEL
LIN {X 0,Y 167.218,Z 464.36,A -85,B 0,C 180,E1 -23182.993,E2 -23182.993} C_VEL
LIN {X 0,Y 166.329,Z 459.956,A -85,B 0,C 180,E1 -23187.68,E2 -23187.68} C_VEL
LIN {X 0,Y 165.358,Z 455.291,A -85,B 0,C 180,E1 -23193.195,E2 -23193.195} C_VEL
LIN {X 0,Y 164.415,Z 451,A -85,B 0,C 180,E1 -23199.023,E2 -23199.023} C_VEL
LIN {X 0,Y 164.486,Z 450.998,A -85,B 0,C 180,E1 -23202.597,E2 -23202.597} C_VEL
LIN {X 0,Y 164.705,Z 450.973,A -85,B 0,C 180,E1 -23208.939,E2 -23208.939} C_VEL
LIN {X 0,Y 164.833,Z 450.957,A -85,B 0,C 180,E1 -23212.651,E2 -23212.651} C_VEL
LIN {X 0,Y 165.052,Z 450.925,A -85,B 0,C 180,E1 -23217.56,E2 -23217.56} C_VEL
LIN {X 0,Y 165.3,Z 450.892,A -85,B 0,C 180,E1 -23220,E2 -23220} C_VEL
LIN {X 0,Y 164.767,Z 450.961,A -85,B 0,C 180,E1 -23224.894,E2 -23224.894} C_VEL
LIN {X 0,Y 164.833,Z 450.949,A -85,B 0,C 180,E1 -23227.349,E2 -23227.349} C_VEL
LIN {X 0,Y 164.705,Z 450.955,A -85,B 0,C 180,E1 -23231.062,E2 -23231.062} C_VEL
LIN {X 0,Y 164.484,Z 450.938,A -85,B 0,C 180,E1 -23237.403,E2 -23237.403} C_VEL
LIN {X 0,Y 164.476,Z 450.98,A -85,B 0,C 180,E1 -23239.989,E2 -23239.989} C_VEL
LIN {X 0,Y 164.395,Z 450.959,A -85,B 0,C 180,E1 -23246.133,E2 -23246.133} C_VEL
LIN {X 0,Y 164.376,Z 450.991,A -85,B 0,C 180,E1 -23251.227,E2 -23251.227} C_VEL
LIN {X 0,Y 164.298,Z 451.015,A -85,B 0,C 180,E1 -23256.789,E2 -23256.789} C_VEL
LIN {X 0,Y 164.312,Z 451.017,A -85,B 0,C 180,E1 -23262.351,E2 -23262.351} C_VEL
LIN {X 0,Y 165.258,Z 453.752,A -85,B 0,C 180,E1 -23263.158,E2 -23263.158} C_VEL
LIN {X 0,Y 167.482,Z 456.813,A -85,B 0,C 180,E1 -23264.49,E2 -23264.49} C_VEL
LIN {X 0,Y 171.828,Z 464.408,A -85,B 0,C 180,E1 -23267.411,E2 -23267.411} C_VEL
LIN {X 0,Y 175.421,Z 471.882,A -85,B 0,C 180,E1 -23270.132,E2 -23270.132} C_VEL
LIN {X 0,Y 178.756,Z 480.477,A -85,B 0,C 180,E1 -23273.192,E2 -23273.192} C_VEL
LIN {X 0,Y 181.495,Z 490.044,A -85,B 0,C 180,E1 -23276.647,E2 -23276.647} C_VEL
LIN {X 0,Y 182.869,Z 497.678,A -85,B 0,C 180,E1 -23279.521,E2 -23279.521} C_VEL
LIN {X 0,Y 182.681,Z 499.137,A -85,B 0,C 180,E1 -23279.991,E2 -23279.991} C_VEL
LIN {X 0,Y 179.517,Z 507.493,A -85,B 0,C 180,E1 -23282.612,E2 -23282.612} C_VEL
LIN {X 0,Y 176.007,Z 515.613,A -85,B 0,C 180,E1 -23285.84,E2 -23285.84} C_VEL
LIN {X 0,Y 173.257,Z 521.649,A -85,B 0,C 180,E1 -23288.904,E2 -23288.904} C_VEL
LIN {X 0,Y 171.058,Z 526.514,A -85,B 0,C 180,E1 -23292.053,E2 -23292.053} C_VEL
LIN {X 0,Y 168.835,Z 530.751,A -85,B 0,C 180,E1 -23295.537,E2 -23295.537} C_VEL
LIN {X 0,Y 167.668,Z 532.984,A -85,B 0,C 180,E1 -23297.902,E2 -23297.902} C_VEL
LIN {X 0,Y 166.682,Z 534.804,A -85,B 0,C 180,E1 -23300.29,E2 -23300.29} C_VEL
LIN {X 0,Y 165.908,Z 536.171,A -85,B 0,C 180,E1 -23302.699,E2 -23302.699} C_VEL
LIN {X 0,Y 165.368,Z 537.691,A -85,B 0,C 180,E1 -23307.564,E2 -23307.564} C_VEL
LIN {X 0,Y 165.295,Z 537.909,A -85,B 0,C 180,E1 -23310,E2 -23310} C_VEL
LIN {X 0,Y 165.367,Z 537.722,A -85,B 0,C 180,E1 -23312.436,E2 -23312.436} C_VEL
LIN {X 0,Y 165.897,Z 536.242,A -85,B 0,C 180,E1 -23317.301,E2 -23317.301} C_VEL
LIN {X 0,Y 166.664,Z 534.907,A -85,B 0,C 180,E1 -23319.711,E2 -23319.711} C_VEL
LIN {X 0,Y 168.272,Z 532.08,A -85,B 0,C 180,E1 -23323.28,E2 -23323.28} C_VEL
LIN {X 0,Y 170.294,Z 528.257,A -85,B 0,C 180,E1 -23326.791,E2 -23326.791} C_VEL
LIN {X 0,Y 172.996,Z 522.326,A -85,B 0,C 180,E1 -23330.871,E2 -23330.871} C_VEL
LIN {X 0,Y 176,Z 515.932,A -85,B 0,C 180,E1 -23334.161,E2 -23334.161} C_VEL
LIN {X 0,Y 179.464,Z 507.886,A -85,B 0,C 180,E1 -23337.396,E2 -23337.396} C_VEL
LIN {X 0,Y 182.565,Z 499.645,A -85,B 0,C 180,E1 -23340.029,E2 -23340.029} C_VEL
LIN {X 0,Y 182.941,Z 498.084,A -85,B 0,C 180,E1 -23340.496,E2 -23340.496} C_VEL
LIN {X 0,Y 181.622,Z 490.321,A -85,B 0,C 180,E1 -23343.418,E2 -23343.418} C_VEL
LIN {X 0,Y 179.062,Z 481.391,A -85,B 0,C 180,E1 -23346.668,E2 -23346.668} C_VEL
LIN {X 0,Y 176.608,Z 474.528,A -85,B 0,C 180,E1 -23349.107,E2 -23349.107} C_VEL
LIN {X 0,Y 172.543,Z 465.713,A -85,B 0,C 180,E1 -23352.31,E2 -23352.31} C_VEL
LIN {X 0,Y 168.684,Z 458.975,A -85,B 0,C 180,E1 -23354.904,E2 -23354.904} C_VEL
LIN {X 0,Y 166.419,Z 455.226,A -85,B 0,C 180,E1 -23356.382,E2 -23356.382} C_VEL
LIN {X 0,Y 164.805,Z 452.851,A -85,B 0,C 180,E1 -23357.392,E2 -23357.392} C_VEL
LIN {X 0,Y 164.325,Z 451.012,A -85,B 0,C 180,E1 -23357.912,E2 -23357.912} C_VEL
LIN {X 0,Y 164.297,Z 451.013,A -85,B 0,C 180,E1 -23363.211,E2 -23363.211} C_VEL
LIN {X 0,Y 164.375,Z 451.005,A -85,B 0,C 180,E1 -23368.773,E2 -23368.773} C_VEL
LIN {X 0,Y 164.418,Z 451.005,A -85,B 0,C 180,E1 -23374.694,E2 -23374.694} C_VEL
LIN {X 0,Y 164.487,Z 450.996,A -85,B 0,C 180,E1 -23380.049,E2 -23380.049} C_VEL
LIN {X 0,Y 164.532,Z 450.991,A -85,B 0,C 180,E1 -23385.15,E2 -23385.15} C_VEL
LIN {X 0,Y 164.769,Z 450.959,A -85,B 0,C 180,E1 -23390.176,E2 -23390.176} C_VEL
LIN {X 0,Y 164.831,Z 450.946,A -85,B 0,C 180,E1 -23392.651,E2 -23392.651} C_VEL
LIN {X 0,Y 165.049,Z 450.924,A -85,B 0,C 180,E1 -23397.559,E2 -23397.559} C_VEL
LIN {X 0,Y 165.299,Z 450.887,A -85,B 0,C 180,E1 -23400,E2 -23400} C_VEL
LIN {X 0,Y 164.767,Z 450.961,A -85,B 0,C 180,E1 -23404.894,E2 -23404.894} C_VEL
LIN {X 0,Y 164.832,Z 450.94,A -85,B 0,C 180,E1 -23407.349,E2 -23407.349} C_VEL
LIN {X 0,Y 164.704,Z 450.967,A -85,B 0,C 180,E1 -23411.062,E2 -23411.062} C_VEL
LIN {X 0,Y 164.484,Z 450.989,A -85,B 0,C 180,E1 -23417.403,E2 -23417.403} C_VEL
LIN {X 0,Y 164.415,Z 451.012,A -85,B 0,C 180,E1 -23420.977,E2 -23420.977} C_VEL
LIN {X 0,Y 165.367,Z 455.393,A -85,B 0,C 180,E1 -23426.812,E2 -23426.812} C_VEL
LIN {X 0,Y 166.013,Z 458.499,A -85,B 0,C 180,E1 -23430.531,E2 -23430.531} C_VEL
LIN {X 0,Y 166.788,Z 462.238,A -85,B 0,C 180,E1 -23434.67,E2 -23434.67} C_VEL
LIN {X 0,Y 167.769,Z 467.545,A -85,B 0,C 180,E1 -23440.045,E2 -23440.045} C_VEL
LIN {X 0,Y 168.203,Z 470.066,A -85,B 0,C 180,E1 -23442.357,E2 -23442.357} C_VEL
LIN {X 0,Y 169.705,Z 473.974,A -85,B 0,C 180,E1 -23443.178,E2 -23443.178} C_VEL
LIN {X 0,Y 171.36,Z 476.76,A -85,B 0,C 180,E1 -23443.985,E2 -23443.985} C_VEL
LIN {X 0,Y 173.414,Z 481.304,A -85,B 0,C 180,E1 -23445.076,E2 -23445.076} C_VEL
LIN {X 0,Y 175.455,Z 486.958,A -85,B 0,C 180,E1 -23446.308,E2 -23446.308} C_VEL
LIN {X 0,Y 176.903,Z 498.685,A -85,B 0,C 180,E1 -23448.306,E2 -23448.306} C_VEL
LIN {X 0,Y 177.399,Z 511.427,A -85,B 0,C 180,E1 -23450.664,E2 -23450.664} C_VEL
LIN {X 0,Y 176.952,Z 523.12,A -85,B 0,C 180,E1 -23453.104,E2 -23453.104} C_VEL
LIN {X 0,Y 175.703,Z 534.805,A -85,B 0,C 180,E1 -23455.945,E2 -23455.945} C_VEL
LIN {X 0,Y 174.201,Z 543.336,A -85,B 0,C 180,E1 -23458.367,E2 -23458.367} C_VEL
LIN {X 0,Y 172.217,Z 552.185,A -85,B 0,C 180,E1 -23461.347,E2 -23461.347} C_VEL
LIN {X 0,Y 170.114,Z 559.503,A -85,B 0,C 180,E1 -23464.292,E2 -23464.292} C_VEL
LIN {X 0,Y 167.232,Z 566.584,A -85,B 0,C 180,E1 -23467.776,E2 -23467.776} C_VEL
LIN {X 0,Y 165.095,Z 572.316,A -85,B 0,C 180,E1 -23471.381,E2 -23471.381} C_VEL
LIN {X 0,Y 163.762,Z 576.88,A -85,B 0,C 180,E1 -23475.079,E2 -23475.079} C_VEL
LIN {X 0,Y 163.177,Z 580.385,A -85,B 0,C 180,E1 -23478.825,E2 -23478.825} C_VEL
LIN {X 0,Y 163.268,Z 582.911,A -85,B 0,C 180,E1 -23482.58,E2 -23482.58} C_VEL
LIN {X 0,Y 163.589,Z 584.051,A -85,B 0,C 180,E1 -23485.071,E2 -23485.071} C_VEL
LIN {X 0,Y 163.996,Z 584.775,A -85,B 0,C 180,E1 -23487.544,E2 -23487.544} C_VEL
LIN {X 0,Y 164.659,Z 585.1,A -85,B 0,C 180,E1 -23490,E2 -23490} C_VEL
LIN {X 0,Y 163.578,Z 584.029,A -85,B 0,C 180,E1 -23494.93,E2 -23494.93} C_VEL
LIN {X 0,Y 163.201,Z 582.614,A -85,B 0,C 180,E1 -23497.92,E2 -23497.92} C_VEL
LIN {X 0,Y 163.285,Z 579.275,A -85,B 0,C 180,E1 -23502.428,E2 -23502.428} C_VEL
LIN {X 0,Y 164.131,Z 575.409,A -85,B 0,C 180,E1 -23506.161,E2 -23506.161} C_VEL
LIN {X 0,Y 165.667,Z 570.436,A -85,B 0,C 180,E1 -23509.839,E2 -23509.839} C_VEL
LIN {X 0,Y 168.639,Z 563.106,A -85,B 0,C 180,E1 -23513.974,E2 -23513.974} C_VEL
LIN {X 0,Y 170.973,Z 556.561,A -85,B 0,C 180,E1 -23516.883,E2 -23516.883} C_VEL
LIN {X 0,Y 173.032,Z 548.638,A -85,B 0,C 180,E1 -23519.839,E2 -23519.839} C_VEL
LIN {X 0,Y 175.031,Z 538.413,A -85,B 0,C 180,E1 -23523.01,E2 -23523.01} C_VEL
LIN {X 0,Y 175.179,Z 537.519,A -85,B 0,C 180,E1 -23523.252,E2 -23523.252} C_VEL
LIN {X 0,Y 175.265,Z 533.122,A -85,B 0,C 180,E1 -23524.529,E2 -23524.529} C_VEL
LIN {X 0,Y 174.413,Z 528.854,A -85,B 0,C 180,E1 -23525.866,E2 -23525.866} C_VEL
LIN {X 0,Y 171.615,Z 518.847,A -85,B 0,C 180,E1 -23528.972,E2 -23528.972} C_VEL
LIN {X 0,Y 171.217,Z 514.066,A -85,B 0,C 180,E1 -23530.153,E2 -23530.153} C_VEL
LIN {X 0,Y 171.138,Z 502.159,A -85,B 0,C 180,E1 -23532.555,E2 -23532.555} C_VEL
LIN {X 0,Y 170.24,Z 491.232,A -85,B 0,C 180,E1 -23534.573,E2 -23534.573} C_VEL
LIN {X 0,Y 169.444,Z 487.923,A -85,B 0,C 180,E1 -23535.266,E2 -23535.266} C_VEL
LIN {X 0,Y 166.062,Z 479.92,A -85,B 0,C 180,E1 -23537.379,E2 -23537.379} C_VEL
LIN {X 0,Y 164.2,Z 475.784,A -85,B 0,C 180,E1 -23538.49,E2 -23538.49} C_VEL
LIN {X 0,Y 163.314,Z 474.095,A -85,B 0,C 180,E1 -23538.992,E2 -23538.992} C_VEL
LIN {X 0,Y 161.315,Z 470.447,A -85,B 0,C 180,E1 -23540.116,E2 -23540.116} C_VEL
LIN {X 0,Y 160.692,Z 468.298,A -85,B 0,C 180,E1 -23540.643,E2 -23540.643} C_VEL
LIN {X 0,Y 159.91,Z 464.039,A -85,B 0,C 180,E1 -23545.156,E2 -23545.156} C_VEL
LIN {X 0,Y 159.15,Z 460.233,A -85,B 0,C 180,E1 -23549.48,E2 -23549.48} C_VEL
LIN {X 0,Y 158.471,Z 456.909,A -85,B 0,C 180,E1 -23553.673,E2 -23553.673} C_VEL
LIN {X 0,Y 157.577,Z 452.758,A -85,B 0,C 180,E1 -23559.491,E2 -23559.491} C_VEL
LIN {X 0,Y 157.426,Z 451.875,A -85,B 0,C 180,E1 -23561.213,E2 -23561.213} C_VEL
LIN {X 0,Y 157.532,Z 451.868,A -85,B 0,C 180,E1 -23567.111,E2 -23567.111} C_VEL
LIN {X 0,Y 157.692,Z 451.848,A -85,B 0,C 180,E1 -23569.731,E2 -23569.731} C_VEL
LIN {X 0,Y 157.77,Z 451.837,A -85,B 0,C 180,E1 -23572.32,E2 -23572.32} C_VEL
LIN {X 0,Y 158.262,Z 451.769,A -85,B 0,C 180,E1 -23580,E2 -23580} C_VEL
LIN {X 0,Y 157.769,Z 451.83,A -85,B 0,C 180,E1 -23587.68,E2 -23587.68} C_VEL
LIN {X 0,Y 157.639,Z 451.832,A -85,B 0,C 180,E1 -23591.237,E2 -23591.237} C_VEL
LIN {X 0,Y 157.444,Z 451.803,A -85,B 0,C 180,E1 -23595.535,E2 -23595.535} C_VEL
LIN {X 0,Y 157.372,Z 451.874,A -85,B 0,C 180,E1 -23600.933,E2 -23600.933} C_VEL
LIN {X 0,Y 157.315,Z 451.835,A -85,B 0,C 180,E1 -23606.684,E2 -23606.684} C_VEL
LIN {X 0,Y 157.277,Z 451.89,A -85,B 0,C 180,E1 -23612.427,E2 -23612.427} C_VEL
LIN {X 0,Y 157.271,Z 451.887,A -85,B 0,C 180,E1 -23616.45,E2 -23616.45} C_VEL
LIN {X 0,Y 157.24,Z 451.891,A -85,B 0,C 180,E1 -23619.335,E2 -23619.335} C_VEL
LIN {X 0,Y 158.317,Z 454.827,A -85,B 0,C 180,E1 -23620.334,E2 -23620.334} C_VEL
LIN {X 0,Y 159.792,Z 456.476,A -85,B 0,C 180,E1 -23621.28,E2 -23621.28} C_VEL
LIN {X 0,Y 162.186,Z 460.554,A -85,B 0,C 180,E1 -23623.038,E2 -23623.038} C_VEL
LIN {X 0,Y 165.249,Z 465.609,A -85,B 0,C 180,E1 -23625.255,E2 -23625.255} C_VEL
LIN {X 0,Y 169.089,Z 473.563,A -85,B 0,C 180,E1 -23628.431,E2 -23628.431} C_VEL
LIN {X 0,Y 172.608,Z 482.683,A -85,B 0,C 180,E1 -23631.955,E2 -23631.955} C_VEL
LIN {X 0,Y 174.941,Z 491.218,A -85,B 0,C 180,E1 -23635.235,E2 -23635.235} C_VEL
LIN {X 0,Y 176.279,Z 498.104,A -85,B 0,C 180,E1 -23637.997,E2 -23637.997} C_VEL
LIN {X 0,Y 176.551,Z 500.159,A -85,B 0,C 180,E1 -23638.835,E2 -23638.835} C_VEL
LIN {X 0,Y 173.308,Z 508.501,A -85,B 0,C 180,E1 -23641.543,E2 -23641.543} C_VEL
LIN {X 0,Y 169.62,Z 516.62,A -85,B 0,C 180,E1 -23644.868,E2 -23644.868} C_VEL
LIN {X 0,Y 166.707,Z 522.674,A -85,B 0,C 180,E1 -23648.045,E2 -23648.045} C_VEL
LIN {X 0,Y 164.387,Z 527.52,A -85,B 0,C 180,E1 -23651.298,E2 -23651.298} C_VEL
LIN {X 0,Y 162.04,Z 531.757,A -85,B 0,C 180,E1 -23654.916,E2 -23654.916} C_VEL
LIN {X 0,Y 160.803,Z 533.99,A -85,B 0,C 180,E1 -23657.377,E2 -23657.377} C_VEL
LIN {X 0,Y 159.759,Z 535.809,A -85,B 0,C 180,E1 -23659.865,E2 -23659.865} C_VEL
LIN {X 0,Y 158.94,Z 537.177,A -85,B 0,C 180,E1 -23662.377,E2 -23662.377} C_VEL
LIN {X 0,Y 158.347,Z 538.696,A -85,B 0,C 180,E1 -23667.456,E2 -23667.456} C_VEL
LIN {X 0,Y 158.268,Z 538.914,A -85,B 0,C 180,E1 -23670,E2 -23670} C_VEL
LIN {X 0,Y 158.346,Z 538.726,A -85,B 0,C 180,E1 -23672.544,E2 -23672.544} C_VEL
LIN {X 0,Y 158.929,Z 537.247,A -85,B 0,C 180,E1 -23677.623,E2 -23677.623} C_VEL
LIN {X 0,Y 159.741,Z 535.912,A -85,B 0,C 180,E1 -23680.136,E2 -23680.136} C_VEL
LIN {X 0,Y 161.44,Z 533.084,A -85,B 0,C 180,E1 -23683.853,E2 -23683.853} C_VEL
LIN {X 0,Y 163.578,Z 529.261,A -85,B 0,C 180,E1 -23687.502,E2 -23687.502} C_VEL
LIN {X 0,Y 166.445,Z 523.333,A -85,B 0,C 180,E1 -23691.731,E2 -23691.731} C_VEL
LIN {X 0,Y 169.612,Z 516.935,A -85,B 0,C 180,E1 -23695.133,E2 -23695.133} C_VEL
LIN {X 0,Y 173.256,Z 508.889,A -85,B 0,C 180,E1 -23698.465,E2 -23698.465} C_VEL
LIN {X 0,Y 176.502,Z 500.65,A -85,B 0,C 180,E1 -23701.174,E2 -23701.174} C_VEL
LIN {X 0,Y 175.778,Z 494.695,A -85,B 0,C 180,E1 -23703.548,E2 -23703.548} C_VEL
LIN {X 0,Y 174.184,Z 488.016,A -85,B 0,C 180,E1 -23706.199,E2 -23706.199} C_VEL
LIN {X 0,Y 171.929,Z 480.607,A -85,B 0,C 180,E1 -23709.043,E2 -23709.043} C_VEL
LIN {X 0,Y 168.585,Z 472.265,A -85,B 0,C 180,E1 -23712.271,E2 -23712.271} C_VEL
LIN {X 0,Y 164.901,Z 464.997,A -85,B 0,C 180,E1 -23715.225,E2 -23715.225} C_VEL
LIN {X 0,Y 160.814,Z 458.303,A -85,B 0,C 180,E1 -23718.205,E2 -23718.205} C_VEL
LIN {X 0,Y 159.745,Z 456.468,A -85,B 0,C 180,E1 -23718.983,E2 -23718.983} C_VEL
LIN {X 0,Y 157.877,Z 454.021,A -85,B 0,C 180,E1 -23720.256,E2 -23720.256} C_VEL
LIN {X 0,Y 157.225,Z 451.904,A -85,B 0,C 180,E1 -23720.96,E2 -23720.96} C_VEL
LIN {X 0,Y 157.28,Z 451.892,A -85,B 0,C 180,E1 -23724.486,E2 -23724.486} C_VEL
LIN {X 0,Y 157.294,Z 451.884,A -85,B 0,C 180,E1 -23728.096,E2 -23728.096} C_VEL
LIN {X 0,Y 157.322,Z 451.882,A -85,B 0,C 180,E1 -23733.466,E2 -23733.466} C_VEL
LIN {X 0,Y 157.397,Z 451.879,A -85,B 0,C 180,E1 -23739.665,E2 -23739.665} C_VEL
LIN {X 0,Y 157.463,Z 451.867,A -85,B 0,C 180,E1 -23744.467,E2 -23744.467} C_VEL
LIN {X 0,Y 157.691,Z 451.838,A -85,B 0,C 180,E1 -23749.731,E2 -23749.731} C_VEL
LIN {X 0,Y 157.768,Z 451.828,A -85,B 0,C 180,E1 -23752.32,E2 -23752.32} C_VEL
LIN {X 0,Y 158.261,Z 451.763,A -85,B 0,C 180,E1 -23760,E2 -23760} C_VEL
LIN {X 0,Y 157.768,Z 451.819,A -85,B 0,C 180,E1 -23767.68,E2 -23767.68} C_VEL
LIN {X 0,Y 157.638,Z 451.845,A -85,B 0,C 180,E1 -23771.237,E2 -23771.237} C_VEL
LIN {X 0,Y 157.455,Z 451.87,A -85,B 0,C 180,E1 -23775.534,E2 -23775.534} C_VEL
LIN {X 0,Y 157.424,Z 451.919,A -85,B 0,C 180,E1 -23779.096,E2 -23779.096} C_VEL
LIN {X 0,Y 158.246,Z 455.984,A -85,B 0,C 180,E1 -23784.955,E2 -23784.955} C_VEL
LIN {X 0,Y 158.993,Z 459.191,A -85,B 0,C 180,E1 -23789.093,E2 -23789.093} C_VEL
LIN {X 0,Y 159.733,Z 462.725,A -85,B 0,C 180,E1 -23793.283,E2 -23793.283} C_VEL
LIN {X 0,Y 160.566,Z 467.654,A -85,B 0,C 180,E1 -23798.587,E2 -23798.587} C_VEL
LIN {X 0,Y 160.727,Z 468.469,A -85,B 0,C 180,E1 -23799.347,E2 -23799.347} C_VEL
LIN {X 0,Y 162.281,Z 472.428,A -85,B 0,C 180,E1 -23800.309,E2 -23800.309} C_VEL
LIN {X 0,Y 163.999,Z 475.139,A -85,B 0,C 180,E1 -23801.243,E2 -23801.243} C_VEL
LIN {X 0,Y 165.802,Z 479.464,A -85,B 0,C 180,E1 -23802.354,E2 -23802.354} C_VEL
LIN {X 0,Y 166.885,Z 481.539,A -85,B 0,C 180,E1 -23802.977,E2 -23802.977} C_VEL
LIN {X 0,Y 169.658,Z 488.5,A -85,B 0,C 180,E1 -23804.766,E2 -23804.766} C_VEL
LIN {X 0,Y 170.418,Z 491.98,A -85,B 0,C 180,E1 -23805.487,E2 -23805.487} C_VEL
LIN {X 0,Y 171.296,Z 504.477,A -85,B 0,C 180,E1 -23807.823,E2 -23807.823} C_VEL
LIN {X 0,Y 171.229,Z 516.122,A -85,B 0,C 180,E1 -23810.225,E2 -23810.225} C_VEL
LIN {X 0,Y 170.322,Z 527.51,A -85,B 0,C 180,E1 -23812.881,E2 -23812.881} C_VEL
LIN {X 0,Y 168.737,Z 538.178,A -85,B 0,C 180,E1 -23815.782,E2 -23815.782} C_VEL
LIN {X 0,Y 167.062,Z 546.021,A -85,B 0,C 180,E1 -23818.274,E2 -23818.274} C_VEL
LIN {X 0,Y 164.988,Z 554.252,A -85,B 0,C 180,E1 -23821.366,E2 -23821.366} C_VEL
LIN {X 0,Y 162.654,Z 561.023,A -85,B 0,C 180,E1 -23824.4,E2 -23824.4} C_VEL
LIN {X 0,Y 159.758,Z 567.636,A -85,B 0,C 180,E1 -23828.042,E2 -23828.042} C_VEL
LIN {X 0,Y 157.731,Z 572.957,A -85,B 0,C 180,E1 -23831.826,E2 -23831.826} C_VEL
LIN {X 0,Y 156.538,Z 577.16,A -85,B 0,C 180,E1 -23835.704,E2 -23835.704} C_VEL
LIN {X 0,Y 156.066,Z 580.329,A -85,B 0,C 180,E1 -23839.623,E2 -23839.623} C_VEL
LIN {X 0,Y 156.183,Z 581.889,A -85,B 0,C 180,E1 -23842.242,E2 -23842.242} C_VEL
LIN {X 0,Y 156.507,Z 583.035,A -85,B 0,C 180,E1 -23844.847,E2 -23844.847} C_VEL
LIN {X 0,Y 156.914,Z 583.761,A -85,B 0,C 180,E1 -23847.433,E2 -23847.433} C_VEL
LIN {X 0,Y 157.579,Z 584.087,A -85,B 0,C 180,E1 -23850,E2 -23850} C_VEL
LIN {X 0,Y 156.495,Z 583.012,A -85,B 0,C 180,E1 -23855.153,E2 -23855.153} C_VEL
LIN {X 0,Y 156.142,Z 581.729,A -85,B 0,C 180,E1 -23858.017,E2 -23858.017} C_VEL
LIN {X 0,Y 156.314,Z 578.252,A -85,B 0,C 180,E1 -23862.992,E2 -23862.992} C_VEL
LIN {X 0,Y 157.234,Z 574.379,A -85,B 0,C 180,E1 -23866.89,E2 -23866.89} C_VEL
LIN {X 0,Y 158.948,Z 569.41,A -85,B 0,C 180,E1 -23870.716,E2 -23870.716} C_VEL
LIN {X 0,Y 162.135,Z 562.083,A -85,B 0,C 180,E1 -23875,E2 -23875} C_VEL
LIN {X 0,Y 164.508,Z 555.517,A -85,B 0,C 180,E1 -23878.03,E2 -23878.03} C_VEL
LIN {X 0,Y 166.666,Z 547.579,A -85,B 0,C 180,E1 -23881.102,E2 -23881.102} C_VEL
LIN {X 0,Y 168.701,Z 537.938,A -85,B 0,C 180,E1 -23884.221,E2 -23884.221} C_VEL
LIN {X 0,Y 170.305,Z 527.179,A -85,B 0,C 180,E1 -23887.124,E2 -23887.124} C_VEL
LIN {X 0,Y 171.096,Z 516.877,A -85,B 0,C 180,E1 -23889.544,E2 -23889.544} C_VEL
LIN {X 0,Y 171.217,Z 514.066,A -85,B 0,C 180,E1 -23890.153,E2 -23890.153} C_VEL
LIN {X 0,Y 170.892,Z 509.219,A -85,B 0,C 180,E1 -23891.29,E2 -23891.29} C_VEL
LIN {X 0,Y 169.778,Z 504.615,A -85,B 0,C 180,E1 -23892.499,E2 -23892.499} C_VEL
LIN {X 0,Y 166.291,Z 495.886,A -85,B 0,C 180,E1 -23895.058,E2 -23895.058} C_VEL
LIN {X 0,Y 163.817,Z 490.083,A -85,B 0,C 180,E1 -23896.801,E2 -23896.801} C_VEL
LIN {X 0,Y 161.264,Z 483.979,A -85,B 0,C 180,E1 -23898.609,E2 -23898.609} C_VEL
LIN {X 0,Y 159.146,Z 479.012,A -85,B 0,C 180,E1 -23900.08,E2 -23900.08} C_VEL
LIN {X 0,Y 157.035,Z 474.617,A -85,B 0,C 180,E1 -23901.488,E2 -23901.488} C_VEL
LIN {X 0,Y 156.301,Z 473.02,A -85,B 0,C 180,E1 -23901.985,E2 -23901.985} C_VEL
LIN {X 0,Y 153.983,Z 469.055,A -85,B 0,C 180,E1 -23903.473,E2 -23903.473} C_VEL
LIN {X 0,Y 153.223,Z 466.656,A -85,B 0,C 180,E1 -23904.135,E2 -23904.135} C_VEL
LIN {X 0,Y 152.301,Z 462.108,A -85,B 0,C 180,E1 -23909.496,E2 -23909.496} C_VEL
LIN {X 0,Y 151.631,Z 458.758,A -85,B 0,C 180,E1 -23913.876,E2 -23913.876} C_VEL
LIN {X 0,Y 150.878,Z 455.409,A -85,B 0,C 180,E1 -23918.689,E2 -23918.689} C_VEL
LIN {X 0,Y 150.364,Z 452.756,A -85,B 0,C 180,E1 -23923.015,E2 -23923.015} C_VEL
LIN {X 0,Y 150.614,Z 452.729,A -85,B 0,C 180,E1 -23929.243,E2 -23929.243} C_VEL
LIN {X 0,Y 150.707,Z 452.717,A -85,B 0,C 180,E1 -23931.958,E2 -23931.958} C_VEL
LIN {X 0,Y 151.222,Z 452.646,A -85,B 0,C 180,E1 -23940,E2 -23940} C_VEL
LIN {X 0,Y 150.707,Z 452.711,A -85,B 0,C 180,E1 -23948.042,E2 -23948.042} C_VEL
LIN {X 0,Y 150.58,Z 452.704,A -85,B 0,C 180,E1 -23951.438,E2 -23951.438} C_VEL
LIN {X 0,Y 150.354,Z 452.685,A -85,B 0,C 180,E1 -23956.288,E2 -23956.288} C_VEL
LIN {X 0,Y 150.354,Z 452.746,A -85,B 0,C 180,E1 -23960.793,E2 -23960.793} C_VEL
LIN {X 0,Y 150.245,Z 452.711,A -85,B 0,C 180,E1 -23967.281,E2 -23967.281} C_VEL
LIN {X 0,Y 150.217,Z 452.771,A -85,B 0,C 180,E1 -23972.632,E2 -23972.632} C_VEL
LIN {X 0,Y 150.246,Z 452.866,A -85,B 0,C 180,E1 -23975.886,E2 -23975.886} C_VEL
LIN {X 0,Y 151.201,Z 455.615,A -85,B 0,C 180,E1 -23976.881,E2 -23976.881} C_VEL
LIN {X 0,Y 153.535,Z 458.274,A -85,B 0,C 180,E1 -23978.616,E2 -23978.616} C_VEL
LIN {X 0,Y 155.321,Z 461.544,A -85,B 0,C 180,E1 -23980.15,E2 -23980.15} C_VEL
LIN {X 0,Y 158.538,Z 466.681,A -85,B 0,C 180,E1 -23982.728,E2 -23982.728} C_VEL
LIN {X 0,Y 162.398,Z 474.395,A -85,B 0,C 180,E1 -23986.177,E2 -23986.177} C_VEL
LIN {X 0,Y 165.284,Z 481.505,A -85,B 0,C 180,E1 -23989.175,E2 -23989.175} C_VEL
LIN {X 0,Y 167.597,Z 488.693,A -85,B 0,C 180,E1 -23992.179,E2 -23992.179} C_VEL
LIN {X 0,Y 169.611,Z 497.7,A -85,B 0,C 180,E1 -23995.968,E2 -23995.968} C_VEL
LIN {X 0,Y 170.101,Z 501.248,A -85,B 0,C 180,E1 -23997.512,E2 -23997.512} C_VEL
LIN {X 0,Y 169.962,Z 502.928,A -85,B 0,C 180,E1 -23998.182,E2 -23998.182} C_VEL
LIN {X 0,Y 165.814,Z 512.421,A -85,B 0,C 180,E1 -24001.521,E2 -24001.521} C_VEL
LIN {X 0,Y 162.113,Z 519.98,A -85,B 0,C 180,E1 -24004.995,E2 -24004.995} C_VEL
LIN {X 0,Y 159.602,Z 525.067,A -85,B 0,C 180,E1 -24007.992,E2 -24007.992} C_VEL
LIN {X 0,Y 156.933,Z 530.075,A -85,B 0,C 180,E1 -24011.73,E2 -24011.73} C_VEL
LIN {X 0,Y 154.64,Z 533.95,A -85,B 0,C 180,E1 -24015.524,E2 -24015.524} C_VEL
LIN {X 0,Y 152.845,Z 536.815,A -85,B 0,C 180,E1 -24019.401,E2 -24019.401} C_VEL
LIN {X 0,Y 151.977,Z 538.182,A -85,B 0,C 180,E1 -24022.025,E2 -24022.025} C_VEL
LIN {X 0,Y 151.327,Z 539.701,A -85,B 0,C 180,E1 -24027.338,E2 -24027.338} C_VEL
LIN {X 0,Y 151.241,Z 539.919,A -85,B 0,C 180,E1 -24030,E2 -24030} C_VEL
LIN {X 0,Y 151.325,Z 539.731,A -85,B 0,C 180,E1 -24032.662,E2 -24032.662} C_VEL
LIN {X 0,Y 151.965,Z 538.251,A -85,B 0,C 180,E1 -24037.975,E2 -24037.975} C_VEL
LIN {X 0,Y 152.827,Z 536.916,A -85,B 0,C 180,E1 -24040.6,E2 -24040.6} C_VEL
LIN {X 0,Y 154.625,Z 534.089,A -85,B 0,C 180,E1 -24044.476,E2 -24044.476} C_VEL
LIN {X 0,Y 156.89,Z 530.265,A -85,B 0,C 180,E1 -24048.274,E2 -24048.274} C_VEL
LIN {X 0,Y 159.936,Z 524.34,A -85,B 0,C 180,E1 -24052.661,E2 -24052.661} C_VEL
LIN {X 0,Y 163.277,Z 517.938,A -85,B 0,C 180,E1 -24056.18,E2 -24056.18} C_VEL
LIN {X 0,Y 167.112,Z 509.891,A -85,B 0,C 180,E1 -24059.614,E2 -24059.614} C_VEL
LIN {X 0,Y 169.826,Z 503.399,A -85,B 0,C 180,E1 -24061.846,E2 -24061.846} C_VEL
LIN {X 0,Y 170.187,Z 501.709,A -85,B 0,C 180,E1 -24062.469,E2 -24062.469} C_VEL
LIN {X 0,Y 169.047,Z 494.461,A -85,B 0,C 180,E1 -24065.594,E2 -24065.594} C_VEL
LIN {X 0,Y 166.84,Z 485.864,A -85,B 0,C 180,E1 -24069.188,E2 -24069.188} C_VEL
LIN {X 0,Y 163.479,Z 476.657,A -85,B 0,C 180,E1 -24073.043,E2 -24073.043} C_VEL
LIN {X 0,Y 159.104,Z 467.74,A -85,B 0,C 180,E1 -24077.03,E2 -24077.03} C_VEL
LIN {X 0,Y 155.567,Z 461.821,A -85,B 0,C 180,E1 -24079.926,E2 -24079.926} C_VEL
LIN {X 0,Y 153.545,Z 458.284,A -85,B 0,C 180,E1 -24081.638,E2 -24081.638} C_VEL
LIN {X 0,Y 151.076,Z 455.351,A -85,B 0,C 180,E1 -24083.511,E2 -24083.511} C_VEL
LIN {X 0,Y 150.24,Z 452.768,A -85,B 0,C 180,E1 -24084.422,E2 -24084.422} C_VEL
LIN {X 0,Y 150.208,Z 452.771,A -85,B 0,C 180,E1 -24089.024,E2 -24089.024} C_VEL
LIN {X 0,Y 150.245,Z 452.761,A -85,B 0,C 180,E1 -24092.718,E2 -24092.718} C_VEL
LIN {X 0,Y 150.354,Z 452.753,A -85,B 0,C 180,E1 -24099.206,E2 -24099.206} C_VEL
LIN {X 0,Y 150.371,Z 452.746,A -85,B 0,C 180,E1 -24103.714,E2 -24103.714} C_VEL
LIN {X 0,Y 150.613,Z 452.716,A -85,B 0,C 180,E1 -24109.242,E2 -24109.242} C_VEL
LIN {X 0,Y 150.706,Z 452.71,A -85,B 0,C 180,E1 -24111.958,E2 -24111.958} C_VEL
LIN {X 0,Y 151.221,Z 452.639,A -85,B 0,C 180,E1 -24120,E2 -24120} C_VEL
LIN {X 0,Y 150.706,Z 452.698,A -85,B 0,C 180,E1 -24128.042,E2 -24128.042} C_VEL
LIN {X 0,Y 150.579,Z 452.722,A -85,B 0,C 180,E1 -24131.438,E2 -24131.438} C_VEL
LIN {X 0,Y 150.362,Z 452.838,A -85,B 0,C 180,E1 -24136.985,E2 -24136.985} C_VEL
LIN {X 0,Y 150.967,Z 455.912,A -85,B 0,C 180,E1 -24141.865,E2 -24141.865} C_VEL
LIN {X 0,Y 151.898,Z 459.925,A -85,B 0,C 180,E1 -24147.56,E2 -24147.56} C_VEL
LIN {X 0,Y 152.875,Z 464.666,A -85,B 0,C 180,E1 -24153.481,E2 -24153.481} C_VEL
LIN {X 0,Y 153.232,Z 466.673,A -85,B 0,C 180,E1 -24155.785,E2 -24155.785} C_VEL
LIN {X 0,Y 154.781,Z 470.677,A -85,B 0,C 180,E1 -24156.909,E2 -24156.909} C_VEL
LIN {X 0,Y 156.862,Z 473.946,A -85,B 0,C 180,E1 -24158.217,E2 -24158.217} C_VEL
LIN {X 0,Y 158.744,Z 478.288,A -85,B 0,C 180,E1 -24159.525,E2 -24159.525} C_VEL
LIN {X 0,Y 159.922,Z 480.649,A -85,B 0,C 180,E1 -24160.303,E2 -24160.303} C_VEL
LIN {X 0,Y 162.46,Z 486.757,A -85,B 0,C 180,E1 -24162.108,E2 -24162.108} C_VEL
LIN {X 0,Y 164.783,Z 492.98,A -85,B 0,C 180,E1 -24163.873,E2 -24163.873} C_VEL
LIN {X 0,Y 165.436,Z 502.965,A -85,B 0,C 180,E1 -24165.881,E2 -24165.881} C_VEL
LIN {X 0,Y 165.322,Z 514.511,A -85,B 0,C 180,E1 -24168.378,E2 -24168.378} C_VEL
LIN {X 0,Y 164.402,Z 525.352,A -85,B 0,C 180,E1 -24170.995,E2 -24170.995} C_VEL
LIN {X 0,Y 162.799,Z 536.029,A -85,B 0,C 180,E1 -24173.971,E2 -24173.971} C_VEL
LIN {X 0,Y 160.804,Z 544.964,A -85,B 0,C 180,E1 -24176.885,E2 -24176.885} C_VEL
LIN {X 0,Y 158.546,Z 553.198,A -85,B 0,C 180,E1 -24180.087,E2 -24180.087} C_VEL
LIN {X 0,Y 156.188,Z 559.995,A -85,B 0,C 180,E1 -24183.258,E2 -24183.258} C_VEL
LIN {X 0,Y 153.494,Z 565.839,A -85,B 0,C 180,E1 -24186.556,E2 -24186.556} C_VEL
LIN {X 0,Y 150.935,Z 571.933,A -85,B 0,C 180,E1 -24190.978,E2 -24190.978} C_VEL
LIN {X 0,Y 149.585,Z 576.133,A -85,B 0,C 180,E1 -24195.024,E2 -24195.024} C_VEL
LIN {X 0,Y 149.031,Z 579.306,A -85,B 0,C 180,E1 -24199.127,E2 -24199.127} C_VEL
LIN {X 0,Y 149.087,Z 580.864,A -85,B 0,C 180,E1 -24201.87,E2 -24201.87} C_VEL
LIN {X 0,Y 149.405,Z 582.015,A -85,B 0,C 180,E1 -24204.602,E2 -24204.602} C_VEL
LIN {X 0,Y 149.833,Z 582.748,A -85,B 0,C 180,E1 -24207.312,E2 -24207.312} C_VEL
LIN {X 0,Y 150.498,Z 583.075,A -85,B 0,C 180,E1 -24210,E2 -24210} C_VEL
LIN {X 0,Y 149.826,Z 582.733,A -85,B 0,C 180,E1 -24212.689,E2 -24212.689} C_VEL
LIN {X 0,Y 149.394,Z 581.992,A -85,B 0,C 180,E1 -24215.399,E2 -24215.399} C_VEL
LIN {X 0,Y 149.087,Z 580.834,A -85,B 0,C 180,E1 -24218.13,E2 -24218.13} C_VEL
LIN {X 0,Y 149.139,Z 578.286,A -85,B 0,C 180,E1 -24222.243,E2 -24222.243} C_VEL
LIN {X 0,Y 149.924,Z 574.752,A -85,B 0,C 180,E1 -24226.336,E2 -24226.336} C_VEL
LIN {X 0,Y 151.533,Z 570.162,A -85,B 0,C 180,E1 -24230.356,E2 -24230.356} C_VEL
LIN {X 0,Y 154.631,Z 563.36,A -85,B 0,C 180,E1 -24234.861,E2 -24234.861} C_VEL
LIN {X 0,Y 157.173,Z 557.279,A -85,B 0,C 180,E1 -24238.003,E2 -24238.003} C_VEL
LIN {X 0,Y 159.904,Z 548.223,A -85,B 0,C 180,E1 -24241.831,E2 -24241.831} C_VEL
LIN {X 0,Y 162.32,Z 537.889,A -85,B 0,C 180,E1 -24245.388,E2 -24245.388} C_VEL
LIN {X 0,Y 164.061,Z 527.725,A -85,B 0,C 180,E1 -24248.309,E2 -24248.309} C_VEL
LIN {X 0,Y 165.073,Z 517.41,A -85,B 0,C 180,E1 -24250.888,E2 -24250.888} C_VEL
LIN {X 0,Y 165.391,Z 505.305,A -85,B 0,C 180,E1 -24253.556,E2 -24253.556} C_VEL
LIN {X 0,Y 164.891,Z 494.45,A -85,B 0,C 180,E1 -24255.738,E2 -24255.738} C_VEL
LIN {X 0,Y 163.954,Z 490.438,A -85,B 0,C 180,E1 -24256.697,E2 -24256.697} C_VEL
LIN {X 0,Y 163.817,Z 490.083,A -85,B 0,C 180,E1 -24256.801,E2 -24256.801} C_VEL
LIN {X 0,Y 162.165,Z 487.691,A -85,B 0,C 180,E1 -24257.773,E2 -24257.773} C_VEL
LIN {X 0,Y 154.61,Z 482.808,A -85,B 0,C 180,E1 -24261.471,E2 -24261.471} C_VEL
LIN {X 0,Y 153.2,Z 480.223,A -85,B 0,C 180,E1 -24262.45,E2 -24262.45} C_VEL
LIN {X 0,Y 152.129,Z 477.76,A -85,B 0,C 180,E1 -24263.296,E2 -24263.296} C_VEL
LIN {X 0,Y 149.992,Z 473.392,A -85,B 0,C 180,E1 -24264.947,E2 -24264.947} C_VEL
LIN {X 0,Y 149.293,Z 471.763,A -85,B 0,C 180,E1 -24265.513,E2 -24265.513} C_VEL
LIN {X 0,Y 146.659,Z 467.694,A -85,B 0,C 180,E1 -24267.479,E2 -24267.479} C_VEL
LIN {X 0,Y 145.624,Z 464.823,A -85,B 0,C 180,E1 -24268.44,E2 -24268.44} C_VEL
LIN {X 0,Y 144.797,Z 460.586,A -85,B 0,C 180,E1 -24274.098,E2 -24274.098} C_VEL
LIN {X 0,Y 143.958,Z 456.681,A -85,B 0,C 180,E1 -24280.017,E2 -24280.017} C_VEL
LIN {X 0,Y 143.328,Z 453.634,A -85,B 0,C 180,E1 -24285.446,E2 -24285.446} C_VEL
LIN {X 0,Y 143.54,Z 453.608,A -85,B 0,C 180,E1 -24288.706,E2 -24288.706} C_VEL
LIN {X 0,Y 143.628,Z 453.597,A -85,B 0,C 180,E1 -24291.559,E2 -24291.559} C_VEL
LIN {X 0,Y 144.18,Z 453.523,A -85,B 0,C 180,E1 -24300,E2 -24300} C_VEL
LIN {X 0,Y 143.628,Z 453.594,A -85,B 0,C 180,E1 -24308.441,E2 -24308.441} C_VEL
LIN {X 0,Y 143.507,Z 453.578,A -85,B 0,C 180,E1 -24311.629,E2 -24311.629} C_VEL
